# B&R Automation Studio project Panasonic_LinkaPowerCP2_A2021055 (part 35)

#### Main.st - Init, cyclic, exit code
```iecst
PROGRAM _INIT
	(* Insert code here *)

END_PROGRAM

PROGRAM _CYCLIC

	//Alarmy pracoviska č.2 (200 - 299)//
	//A200 - ST3_Zakladanie tesnenia - porucha precitania kodu paletky !!!
	//A201 - ST3_Zakladanie tesnenia - porucha precitania QR kodu !!!
	//A202 - ST3_Zakladanie tesnenia - porucha serva zdvihu !!!
	//A203 - ST3_Zakladanie tesnenia - porucha serva pojazdu !!!
	//A204 - ST3_Zakladanie tesnenia - porucha vysunutia pritlacania !!!
	//A205 - ST3_Zakladanie tesnenia - porucha zasunutia pritlacania !!!
	//A206 - ST3_Zakladanie tesnenia - narusenie optickej bariery !!!
	//A207 - ST3_Zakladanie tesnenia - bol stlaceny bumper suflika !!!
	//A208 - ST3_Zakladanie tesnenia - porucha snimaca kopita IS7 !!!
	//A209 - ST4_Maticovacka - porucha vysunutia centrovacky !!!
	//A210 - ST4_Maticovacka - porucha zasunutia centrovacky !!!
	//A211 - ST4_Maticovacka - porucha precitania kodu paletky !!!
	//A212 - ST5_Srobovanie - porucha vysunutia centrovacky !!!
	//A213 - ST5_Srobovanie - porucha zasunutia centrovacky !!!
	//A214 - ST5_Srobovanie - porucha precitania kodu paletky !!!
	//A215 - ST5_Srobovanie - porucha serva manipulatora os X !!!
	//A216 - ST5_Srobovanie - porucha serva manipulatora os Y !!!
	//A217 - ST6_Zvaranie - porucha vysunutia centrovacky !!!
	//A218 - ST6_Zvaranie - porucha zasunutia centrovacky !!!
	//A219 - ST6_Zvaranie - porucha precitania kodu paletky !!!
	//A220 - ST6_Zvaranie - porucha serva zdvihu zvarania !!!
	//A221 - ST6_Zvaranie - porucha presunu pojazdu zvarania !!!
	//A222 - ST6_Zvaranie - porucha zvaracky !!!
	//A223 - ST6_Cistenie - porucha zatvorenia dveri !!!
	//A224 - ST6_Cistenie - porucha otvorenia dveri !!!
	//A225 - ST3_Zakladanie tesnenia - CAM 1 porucha komunikacie FTP !!!
	//A226 - ST3_Zakladanie tesnenia - CAM 7 porucha komunikacie FTP !!!
	//A227 - ST3_Zakladanie tesnenia - CAM 8 porucha komunikacie FTP !!!
	//A228 - ST3_Zakladanie tesnenia - CAM 17 porucha komunikacie FTP !!!
	//A229 - ST4_Maticovacka - CAM 9 porucha komunikacie FTP !!!
	//A230 - ST3_Zakladanie tesnenia - porucha komunikacie zo serverom !!!
	//A231 - ST4_Maticovacka - porucha komunikacie zo serverom !!!
	//A232 - ST5_Srobovanie - CAM 10 porucha komunikacie FTP !!!
	//A233 - ST5_Srobovanie - porucha komunikacie zo serverom !!!
	//A234 - ST6_Zvaranie - CAM 11 porucha komunikacie FTP !!!
	//A235 - ST6_Zvaranie - CAM 12 porucha komunikacie FTP !!!
	//A236 - ST6_Zvaranie - porucha komunikacie zo serverom !!!
	//A237 - ST5_Srobovanie - skrutka M4 nieje pripravena !!!
	//A238 - ST5_Srobovanie - skrutka M5 nieje pripravena !!!
	//A239 - ST5_Srobovanie - skrutka M6 nieje pripravena !!!
	//A240 - ST4_Maticovacka - matica M4 nieje pripravena !!!
	//A241 - ST5_Srobovanie - porucha serva manipulatora os X !!!
	//A242 - ST5_Srobovanie - porucha serva manipulatora os Y !!!
	//A243 - P2_Robot - porucha napajania !!!
	//A244 - P2_Robot - nieje online !!!
	//A245 - Pracovisko 2 - Porucha tlaku vzduchu !!!
	//A246 - Pracovisko 2 - Modul DI21 nieje online !!!
	//A247 - Pracovisko 2 - Modul DI22 nieje online !!!
	//A248 - Pracovisko 2 - Modul DI23 nieje online !!!
	//A249 - Pracovisko 2 - Modul DI24 nieje online !!!
	//A250 - Pracovisko 2 - Modul DI25 nieje online !!!
	//A251 - Pracovisko 2 - Modul DM21 nieje online !!!
	//A252 - Pracovisko 2 - Modul DS21 nieje online !!!
    //A253 - Pracovisko 2 - Modul DS22 nieje online !!!
    //A254 - Pracovisko 2 - Modul DS23 nieje online !!!
	//A255 - Pracovisko 2 - Modul SI21 nieje online !!!
    //A256 - Pracovisko 2 - Modul SI22 nieje online !!!
	//A257 - Pracovisko 2 - Ventilovy termnal VT1 nieje online !!!
	//A258 - Pracovisko 2 - Ventilovy termnal VT2 nieje online !!!
    //A259 - Pracovisko 2 - Ventilovy termnal VT3 nieje online !!!
    //A260 - ST5_Srobovanie - Skrutkovacka M4 nieje online !!!
    //A261 - ST5_Srobovanie - Skrutkovacka M5 nieje online !!!
    //A262 - ST5_Srobovanie - Skrutkovacka M6 nieje online !!!
    //A263 - ST4_Maticovacka - Maticovacka M4 nieje online !!!
    //A264 - Pracovisko 2 - Kamery KAM1, KAM7, KAM10, KAM11, KAM12 a KAM17 niesu online !!!
    //A265 - Pracovisko 2 - Kamera KAM8 nieje online !!!
    //A266 - Pracovisko 2 - Kamera KAM9 nieje online !!!
    //A267 - ST4_Maticovacka - Porucha maticovacky M4 !!!
    //A268 - ST5_Srobovanie - Porucha vysunutia skrutkovacky M4 !!!
    //A269 - ST5_Srobovanie - Porucha vysunutia skrutkovacky M5 !!!
    //A270 - ST5_Srobovanie - Porucha vysunutia skrutkovacky M6 !!!
    //A271 - P2_Robot - porucha !!!
    //A272 - ST5_Srobovanie - Presiahnuty cas skrutkovania skrutky M4 !!!
    //A273 - ST5_Srobovanie - Presiahnuty cas skrutkovania skrutky M5 !!!
    //A274 - ST5_Srobovanie - Presiahnuty cas skrutkovania skrutky M6 !!!
    //A275 - ST5_Srobovanie - Skrutkovacka M4 nieje READY !!!
    //A276 - ST5_Srobovanie - Skrutkovacka M5 nieje READY !!!
    //A277 - ST5_Srobovanie - Skrutkovacka M6 nieje READY !!!
    //A278 - Pracovisko 2 - Prekrocena teplota motora vrchneho dopravnika !!!
    //A279 - Pracovisko 2 - Prekrocena teplota motora spodneho dopravnika !!!
    //A280 - Pracovisko 2 - Narusenie optickej bariery na vystupe !!!
    //A281 - Pracovisko 2 - Bolo stlacene tlacitko CS na ovladacom paneli !!!
    //A282 - Pracovisko 2 - Bolo stlacene tlacitko CS na rozvodnej skrini !!!
    //A283 - Pracovisko 2 - Bolo stlacene tlacitko CS robota !!!
    //A284 - Pracovisko 2 - Bolo stlacene tlacitko CS na dvojrucnom ovladani !!!
    //A285 - P2_Robot - Porucha odobratia Top Coveru z paletky !!!
    //A286 - ST3_Zakladanie tesnenia - Porucha vyvezenia paletky zo stopra !!!
    //A287 - ST4_Maticovacka - Porucha vyvezenia paletky zo stopra !!!
	//A288 - ST5_Srobovanie - Porucha vyvezenia paletky zo stopra !!!
    //A289 - ST6_Zvaranie - Porucha vyvezenia paletky zo stopra !!!
    //A290 - ST3_Zakladanie tesnenia - Porucha komunikacie s kamerou CAM 1 !!!
    //A291 - ST3_Zakladanie tesnenia - Porucha komunikacie s kamerou CAM 7 !!!
    //A292 - ST3_Zakladanie tesnenia - Porucha komunikacie s kamerou CAM 8 !!!
    //A293 - ST3_Zakladanie tesnenia - Porucha komunikacie s kamerou CAM 17 !!!
    //A294 - ST4_Maticovacka - Porucha komunikacie s kamerou CAM 9 !!!
    //A295 - ST5_Srobovanie - Porucha komunikacie s kamerou CAM 10 !!!
    //A296 - ST6_Zvaranie - Porucha komunikacie s kamerou CAM 11 !!!
    //A297 - ST6_Zvaranie - Porucha komunikacie s kamerou CAM 12 !!!
    //A298 - ST4_Maticovacka - Porucha pripravy matice M4 !!!
    //A299 - Akumulacny stoper - Porucha vyvezenia paletky zo stopra !!!

    //*********************Pracovisko 2 - Porucha tlaku vzduchu*********************************//
	IF CasKontroly_TlakVzduchu.Q THEN
		P2_Alarmy[245]:= TRUE;
		P2_Pracovisko.STAV.Porucha_ST1:= TRUE;
		P2_Pracovisko.STAV.Porucha_ST2:= TRUE;
		P2_Pracovisko.STAV.Porucha_ST3:= TRUE;
		P2_Pracovisko.STAV.Porucha_ST4:= TRUE;
		P2_Pracovisko.STAV.Porucha_ST5:= TRUE;
	END_IF

	IF Safety.STAV.P2_ZonaBunky_AKTIVNA AND NOT P2_Pracovisko.IN.TlakVzduchu_OK THEN
		CasKontroly_TlakVzduchu.IN:= TRUE;
	ELSE
		CasKontroly_TlakVzduchu.IN:= FALSE;
	END_IF

	CasKontroly_TlakVzduchu.PT:= T#5s;
	CasKontroly_TlakVzduchu();

	//**********************************Porucha - kamerovy systém nieje online****************************************//
	IF CasKontroly_KAMsystem.Q THEN
		P2_Alarmy[264]:= TRUE;
		P2_Pracovisko.STAV.Porucha_ST1:= TRUE;
		P2_Pracovisko.STAV.Porucha_ST2:= TRUE;
		P2_Pracovisko.STAV.Porucha_ST3:= TRUE;
		P2_Pracovisko.STAV.Porucha_ST4:= TRUE;
		P2_Pracovisko.STAV.Porucha_ST5:= TRUE;
	END_IF

	IF CasKontroly_KAM8.Q THEN
		P2_Alarmy[265]:= TRUE;
		P2_Pracovisko.STAV.Porucha_ST1:= TRUE;
	END_IF

	IF CasKontroly_KAM9.Q THEN
		P2_Alarmy[266]:= TRUE;
		P2_Pracovisko.STAV.Porucha_ST2:= TRUE;
	END_IF

	IF NOT P3_Pracovisko.IN.Kamery_ControlUnit_KomOK AND P2_Pracovisko.Automat THEN
		CasKontroly_KAMsystem.IN:= TRUE;
	ELSE
		CasKontroly_KAMsystem.IN:= FALSE;
	END_IF

	IF NOT CAM8.STAV.READY AND P2_Pracovisko.Automat THEN
		CasKontroly_KAM8.IN:= TRUE;
	ELSE
		CasKontroly_KAM8.IN:= FALSE;
	END_IF

	IF NOT CAM9.STAV.READY AND P2_Pracovisko.Automat THEN
		CasKontroly_KAM9.IN:= TRUE;
	ELSE
		CasKontroly_KAM9.IN:= FALSE;
	END_IF

	CasKontroly_KAMsystem.PT:= T#2s;
	CasKontroly_KAMsystem();
    CasKontroly_KAM8.PT:= T#2s;
	CasKontroly_KAM8();
	CasKontroly_KAM9.PT:= T#2s;
	CasKontroly_KAM9();

	//**********************************Porucha - IO moduly niesu online**************************************************//
	IF CasKontroly_Moduly.Q THEN
		P2_Alarmy[246]:= TRUE;
		P2_Pracovisko.STAV.Porucha_ST1:= TRUE;
		P2_Pracovisko.STAV.Porucha_ST2:= TRUE;
		P2_Pracovisko.STAV.Porucha_ST3:= TRUE;
		P2_Pracovisko.STAV.Porucha_ST4:= TRUE;
		P2_Pracovisko.STAV.Porucha_ST5:= TRUE;
	END_IF

	IF Safety.STAV.P2_ZonaBunky_AKTIVNA AND (NOT P2_Pracovisko.IN.ModulFesto_IO_KomOK OR NOT P2_Pracovisko.IN.ModulWeidmuller_IO_KomOK) THEN
		CasKontroly_Moduly.IN:= TRUE;
	ELSE
		CasKontroly_Moduly.IN:= FALSE;
	END_IF

	CasKontroly_Moduly.PT:= T#2s;
	CasKontroly_Moduly();

	//********************************Porucha - ventilového terminálu*********************************************//
	IF CasKontroly_VentTerminalov.Q THEN
		P2_Alarmy[257]:= TRUE;
		P2_Pracovisko.STAV.Porucha_ST1:= TRUE;
		P2_Pracovisko.STAV.Porucha_ST2:= TRUE;
		P2_Pracovisko.STAV.Porucha_ST3:= TRUE;
		P2_Pracovisko.STAV.Porucha_ST4:= TRUE;
		P2_Pracovisko.STAV.Porucha_ST5:= TRUE;
	END_IF

	IF Safety.STAV.P2_ZonaBunky_AKTIVNA AND NOT P2_Pracovisko.IN.VentilovyTerminal_KomOK THEN
		CasKontroly_VentTerminalov.IN:= TRUE;
	ELSE
		CasKontroly_VentTerminalov.IN:= FALSE;
	END_IF

	CasKontroly_VentTerminalov.PT:= T#2s;
	CasKontroly_VentTerminalov();

	//********************************Porucha - skrutkovacky niesu online**********************************************//
	IF CasKontroly_Skrutkovacky.Q THEN
		IF NOT P2_Pracovisko.IN.Skrutkovacka_M4_KomOK THEN
			P2_Alarmy[260]:= TRUE;
			P2_Pracovisko.STAV.Porucha_ST4:= TRUE;
		END_IF
		IF NOT P2_Pracovisko.IN.Skrutkovacka_M5_KomOK THEN
			P2_Alarmy[261]:= TRUE;
			P2_Pracovisko.STAV.Porucha_ST4:= TRUE;
		END_IF
		IF NOT P2_Pracovisko.IN.Skrutkovacka_M6_KomOK THEN
			P2_Alarmy[262]:= TRUE;
			P2_Pracovisko.STAV.Porucha_ST4:= TRUE;
		END_IF
		IF NOT P2_Pracovisko.IN.Maticovacka_M4_KomOK THEN
			P2_Alarmy[263]:= TRUE;
			P2_Pracovisko.STAV.Porucha_ST2:= TRUE;
		END_IF
	END_IF

	IF Safety.STAV.P2_ZonaBunky_AKTIVNA AND
		(NOT P2_Pracovisko.IN.Skrutkovacka_M4_KomOK OR
		NOT P2_Pracovisko.IN.Skrutkovacka_M5_KomOK OR
		NOT P2_Pracovisko.IN.Skrutkovacka_M6_KomOK OR
		NOT P2_Pracovisko.IN.Maticovacka_M4_KomOK) THEN
		CasKontroly_Skrutkovacky.IN:= TRUE;
	ELSE
		CasKontroly_Skrutkovacky.IN:= FALSE;
	END_IF

	CasKontroly_Skrutkovacky.PT:= T#2s;
	CasKontroly_Skrutkovacky();

	//*********************************Porucha - robot nieje online************************************************//
	IF CasKontroly_Robota.Q THEN
		P2_Alarmy[244]:= TRUE;
		P2_Pracovisko.STAV.Porucha_ST4:= TRUE;
		P2_Pracovisko.STAV.Porucha_ST5:= TRUE;
	END_IF

	IF Safety.STAV.P2_ZonaBunky_AKTIVNA AND NOT P2_Pracovisko.IN.Robot_KomOK THEN
		CasKontroly_Robota.IN:= TRUE;
	ELSE
		CasKontroly_Robota.IN:= FALSE;
	END_IF

	CasKontroly_Robota.PT:= T#2s;
	CasKontroly_Robota();

	//********************Pracovisko 2 - Porucha ochrannej bariéry zdvihu zakladača tesnenia****************************************//
	IF CasKontroly_BarieryZakladaca.Q THEN
		P2_Alarmy[206]:= TRUE;
		P2_Pracovisko.STAV.Porucha_ST1:= TRUE;
	END_IF

    CasKontroly_BarieryZakladaca.IN:= P2_ZakladacTesnenia.Automat AND NOT Safety.STAV.P2_ZaklTesn_Bariera_AKTIVNA AND Safety.STAV.P2_ZaklTesn_PojazdMuting_AKTIVNY;
	CasKontroly_BarieryZakladaca.PT:= T#2s;
	CasKontroly_BarieryZakladaca();

	//*********************Pracovisko 2 - Porucha serva zdvihu zakladača tesnenia***************//
	IF CasPoruchyServaZdvihuZakladaca.Q THEN
		P2_Alarmy[202]:= TRUE;
		P2_Pracovisko.STAV.Porucha_ST1:= TRUE;
	END_IF

	IF Safety.STAV.P2_ZonaZakladacaZdvih_AKTIVNA AND P2_ZakladacTesnenia.ServoZdvihuZakladaca.Status.Error THEN
		CasPoruchyServaZdvihuZakladaca.IN:= TRUE;
	ELSE
		CasPoruchyServaZdvihuZakladaca.IN:= FALSE;
	END_IF

	CasPoruchyServaZdvihuZakladaca.PT:= T#2s;
	CasPoruchyServaZdvihuZakladaca();

	//********************Pracovisko 2 - Porucha bumpera suflíka zakladača tesnenia****************************************//
	IF P2_ZakladacTesnenia.Automat AND NOT Safety.STAV.P2_ZaklTesn_Bumper_AKTIVNY THEN
		P2_Alarmy[207]:= TRUE;
		P2_Pracovisko.STAV.Porucha_ST1:= TRUE;
	END_IF

	//*********************Pracovisko 2 - Porucha serva pojazdu zakladača tesnenia***************//
	IF CasPoruchyServaPojazduZakladaca.Q THEN
		P2_Alarmy[203]:= TRUE;
		P2_Pracovisko.STAV.Porucha_ST1:= TRUE;
	END_IF

	IF Safety.STAV.P2_ZonaZakladacaPojazd_AKTIVNA AND P2_ZakladacTesnenia.ServoPojazduZakladaca.Status.Error THEN
		CasPoruchyServaPojazduZakladaca.IN:= TRUE;
	ELSE
		CasPoruchyServaPojazduZakladaca.IN:= FALSE;
	END_IF

	CasPoruchyServaPojazduZakladaca.PT:= T#2s;
	CasPoruchyServaPojazduZakladaca();

	//*********************Pracovisko 2 - Porucha serva manipulatora šrobovania os X***************//
	IF CasPoruchyServaSrobovaniaOsX.Q THEN
		P2_Alarmy[215]:= TRUE;
		P2_Pracovisko.STAV.Porucha_ST4:= TRUE;
	END_IF

	IF Safety.STAV.P2_ZonaBunky_AKTIVNA AND P2_Srobovanie.ServoManipulOsX.Status.Error THEN
		CasPoruchyServaSrobovaniaOsX.IN:= TRUE;
	ELSE
		CasPoruchyServaSrobovaniaOsX.IN:= FALSE;
	END_IF

	CasPoruchyServaSrobovaniaOsX.PT:= T#2s;
	CasPoruchyServaSrobovaniaOsX();

	//*********************Pracovisko 2 - Porucha serva manipulatora šrobovania os Y***************//
	IF CasPoruchyServaSrobovaniaOsY.Q THEN
		P2_Alarmy[216]:= TRUE;
		P2_Pracovisko.STAV.Porucha_ST4:= TRUE;
	END_IF

	IF Safety.STAV.P2_ZonaBunky_AKTIVNA AND P2_Srobovanie.ServoManipulOsY.Status.Error THEN
		CasPoruchyServaSrobovaniaOsY.IN:= TRUE;
	ELSE
		CasPoruchyServaSrobovaniaOsY.IN:= FALSE;
	END_IF

	CasPoruchyServaSrobovaniaOsY.PT:= T#2s;
	CasPoruchyServaSrobovaniaOsY();

	//*********************Pracovisko 2 - Porucha serva manipulatora šrobovania os Z M4***************//
	IF CasPoruchyServaSrobovaniaOsZ_M4.Q THEN
		P2_Alarmy[247]:= TRUE;
		P2_Pracovisko.STAV.Porucha_ST4:= TRUE;
	END_IF

	IF Safety.STAV.P1_ZonaBunky_AKTIVNA AND P1_Srobovanie.ServoManipulOsZ_M4.Status.Error THEN
		CasPoruchyServaSrobovaniaOsZ_M4.IN:= TRUE;
	ELSE
		CasPoruchyServaSrobovaniaOsZ_M4.IN:= FALSE;
	END_IF

	CasPoruchyServaSrobovaniaOsZ_M4.PT:= T#2s;
	CasPoruchyServaSrobovaniaOsZ_M4();

	//**********************Pracovisko 2 - Porucha serva zdvihu zvarania****************************//
	IF CasPoruchyServaZdvihuZvarania.Q THEN
		P2_Alarmy[220]:= TRUE;
		P2_Pracovisko.STAV.Porucha_ST5:= TRUE;
	END_IF

	IF Safety.STAV.P2_ZonaBunky_AKTIVNA AND P2_Zvaranie.ServoZdvihuZvarania.Status.Error THEN
		CasPoruchyServaZdvihuZvarania.IN:= TRUE;
	ELSE
		CasPoruchyServaZdvihuZvarania.IN:= FALSE;
	END_IF

	CasPoruchyServaZdvihuZvarania.PT:= T#2s;
	CasPoruchyServaZdvihuZvarania();

	//********************Pracovisko 2 - Porucha skrutkovacieho setu M4******************************//
	IF P2_Srobovanie.Automat AND P2_Srobovanie.SkrutSet_M4.STAV.ERROR THEN
		P2_Alarmy[248]:= TRUE;
		P2_Pracovisko.STAV.Porucha_ST4:= TRUE;
	END_IF

	//********************Pracovisko 2 - Porucha skrutkovacieho setu matice M4******************************//
	IF P2_StoperMaticovacky.Automat AND P2_StoperMaticovacky.SkrutSet_MaticaM4.STAV.ERROR THEN
		P2_Alarmy[249]:= TRUE;
		P2_Pracovisko.STAV.Porucha_ST2:= TRUE;
	END_IF

	//****************************Pracovisko 2 - porucha vrchného dopravníka**********************************//
	IF NOT P2_Dopravniky.IN.TeplotaMotoraDopravBunky_OK AND P2_Pracovisko.STAV.Automat THEN
		P2_Alarmy[278]:= TRUE;
		P2_Pracovisko.STAV.Porucha_ST1:= TRUE;
		P2_Pracovisko.STAV.Porucha_ST2:= TRUE;
		P2_Pracovisko.STAV.Porucha_ST3:= TRUE;
		P2_Pracovisko.STAV.Porucha_ST4:= TRUE;
		P2_Pracovisko.STAV.Porucha_ST5:= TRUE;
	END_IF

	//*****************************Pracovisko 2 - porucha spodného dopravníka************************************//
	IF NOT P2_Dopravniky.IN.TeplotaMotoraVratnehoDoprav_OK AND P2_Pracovisko.STAV.Automat THEN
		P2_Alarmy[279]:= TRUE;
	END_IF

	//******************************Pracovisko 2 - narušenie výstupnej bariery***********************************//
	IF NOT Safety.STAV.P3_Bunka_VstupBariera_AKTIVNA AND NOT Safety.STAV.P3_Bunka_Zamky_AKTIVNE AND NOT Safety.STAV.P3_VyblokovanieZamkov_AKTIVNE AND P2_Pracovisko.STAV.Automat THEN
		P2_Alarmy[280]:= TRUE;
		P2_Pracovisko.STAV.Porucha_ST2:= TRUE;
		P2_Pracovisko.STAV.Porucha_ST3:= TRUE;
		P2_Pracovisko.STAV.Porucha_ST4:= TRUE;
		P2_Pracovisko.STAV.Porucha_ST5:= TRUE;
	END_IF

	//******************************Stlačenie tlačítok CS*******************************************************//
	IF EDGENEG(Safety.STAV.P2_Panel_TlacitkoCS_ODBLOK) THEN
		P2_Alarmy[281]:= TRUE;
	END_IF

	IF EDGENEG(Safety.STAV.P2_Rozvadzac_TlacitkoCS_ODBLOK) THEN
		P2_Alarmy[282]:= TRUE;
	END_IF

	IF EDGENEG(Safety.STAV.P2_Robot_TlacitkoCS_ODBLOK) THEN
		P2_Alarmy[283]:= TRUE;
	END_IF

	IF EDGENEG(Safety.STAV.P2_DvojrucOvl_TlacitkoCS_ODBLOK) THEN
		P2_Alarmy[284]:= TRUE;
	END_IF

	//***************************************************Nasetovanie alarmov****************************************************//

	IF P2_Alarmy[200] THEN
		MpAlarmXSet(gAlarmXCore, 'A200');
	ELSE
		MpAlarmXReset(gAlarmXCore, 'A200');
	END_IF

	IF P2_Alarmy[201] THEN
		MpAlarmXSet(gAlarmXCore, 'A201');
	ELSE
		MpAlarmXReset(gAlarmXCore, 'A201');
	END_IF

	IF P2_Alarmy[202] THEN
		MpAlarmXSet(gAlarmXCore, 'A202');
	ELSE
		MpAlarmXReset(gAlarmXCore, 'A202');
	END_IF

	IF P2_Alarmy[203] THEN
		MpAlarmXSet(gAlarmXCore, 'A203');
	ELSE
		MpAlarmXReset(gAlarmXCore, 'A203');
	END_IF

	IF P2_Alarmy[204] THEN
		MpAlarmXSet(gAlarmXCore, 'A204');
	ELSE
		MpAlarmXReset(gAlarmXCore, 'A204');
	END_IF

	IF P2_Alarmy[205] THEN
		MpAlarmXSet(gAlarmXCore, 'A205');
	ELSE
		MpAlarmXReset(gAlarmXCore, 'A205');
	END_IF

	IF P2_Alarmy[206] THEN
		MpAlarmXSet(gAlarmXCore, 'A206');
	ELSE
		MpAlarmXReset(gAlarmXCore, 'A206');
	END_IF

	IF P2_Alarmy[207] THEN
		MpAlarmXSet(gAlarmXCore, 'A207');
	ELSE
		MpAlarmXReset(gAlarmXCore, 'A207');
	END_IF

	IF P2_Alarmy[208] THEN
		MpAlarmXSet(gAlarmXCore, 'A208');
	ELSE
		MpAlarmXReset(gAlarmXCore, 'A208');
	END_IF

	IF P2_Alarmy[209] THEN
		MpAlarmXSet(gAlarmXCore, 'A209');
	ELSE
		MpAlarmXReset(gAlarmXCore, 'A209');
	END_IF

	IF P2_Alarmy[210] THEN
		MpAlarmXSet(gAlarmXCore, 'A210');
	ELSE
		MpAlarmXReset(gAlarmXCore, 'A210');
	END_IF

	IF P2_Alarmy[211] THEN
		MpAlarmXSet(gAlarmXCore, 'A211');
	ELSE
		MpAlarmXReset(gAlarmXCore, 'A211');
	END_IF

	IF P2_Alarmy[212] THEN
		MpAlarmXSet(gAlarmXCore, 'A212');
	ELSE
		MpAlarmXReset(gAlarmXCore, 'A212');
	END_IF

	IF P2_Alarmy[213] THEN
		MpAlarmXSet(gAlarmXCore, 'A213');
	ELSE
		MpAlarmXReset(gAlarmXCore, 'A213');
	END_IF

	IF P2_Alarmy[214] THEN
		MpAlarmXSet(gAlarmXCore, 'A214');
	ELSE
		MpAlarmXReset(gAlarmXCore, 'A214');
	END_IF

	IF P2_Alarmy[215] THEN
		MpAlarmXSet(gAlarmXCore, 'A215');
	ELSE
		MpAlarmXReset(gAlarmXCore, 'A215');
	END_IF

	IF P2_Alarmy[216] THEN
		MpAlarmXSet(gAlarmXCore, 'A216');
	ELSE
		MpAlarmXReset(gAlarmXCore, 'A216');
	END_IF

	IF P2_Alarmy[217] THEN
		MpAlarmXSet(gAlarmXCore, 'A217');
	ELSE
		MpAlarmXReset(gAlarmXCore, 'A217');
	END_IF

	IF P2_Alarmy[218] THEN
		MpAlarmXSet(gAlarmXCore, 'A218');
	ELSE
		MpAlarmXReset(gAlarmXCore, 'A218');
	END_IF

	IF P2_Alarmy[219] THEN
		MpAlarmXSet(gAlarmXCore, 'A219');
	ELSE
		MpAlarmXReset(gAlarmXCore, 'A219');
	END_IF

	IF P2_Alarmy[220] THEN
		MpAlarmXSet(gAlarmXCore, 'A220');
	ELSE
		MpAlarmXReset(gAlarmXCore, 'A220');
	END_IF

	IF P2_Alarmy[221] THEN
		MpAlarmXSet(gAlarmXCore, 'A221');
	ELSE
		MpAlarmXReset(gAlarmXCore, 'A221');
	END_IF

	IF P2_Alarmy[222] THEN
		MpAlarmXSet(gAlarmXCore, 'A222');
	ELSE
		MpAlarmXReset(gAlarmXCore, 'A222');
	END_IF

	IF P2_Alarmy[223] THEN
		MpAlarmXSet(gAlarmXCore, 'A223');
	ELSE
		MpAlarmXReset(gAlarmXCore, 'A223');
	END_IF

	IF P2_Alarmy[224] THEN
		MpAlarmXSet(gAlarmXCore, 'A224');
	ELSE
		MpAlarmXReset(gAlarmXCore, 'A224');
	END_IF

	IF P2_Alarmy[225] THEN
		MpAlarmXSet(gAlarmXCore, 'A225');
	ELSE
		MpAlarmXReset(gAlarmXCore, 'A225');
	END_IF

	IF P2_Alarmy[226] THEN
		MpAlarmXSet(gAlarmXCore, 'A226');
	ELSE
		MpAlarmXReset(gAlarmXCore, 'A226');
	END_IF

	IF P2_Alarmy[227] THEN
		MpAlarmXSet(gAlarmXCore, 'A227');
	ELSE
		MpAlarmXReset(gAlarmXCore, 'A227');
	END_IF

	IF P2_Alarmy[228] THEN
		MpAlarmXSet(gAlarmXCore, 'A228');
	ELSE
		MpAlarmXReset(gAlarmXCore, 'A228');
	END_IF

	IF P2_Alarmy[229] THEN
		MpAlarmXSet(gAlarmXCore, 'A229');
	ELSE
		MpAlarmXReset(gAlarmXCore, 'A229');
	END_IF

	IF P2_Alarmy[230] THEN
		MpAlarmXSet(gAlarmXCore, 'A230');
	ELSE
		MpAlarmXReset(gAlarmXCore, 'A230');
	END_IF

	IF P2_Alarmy[231] THEN
		MpAlarmXSet(gAlarmXCore, 'A231');
	ELSE
		MpAlarmXReset(gAlarmXCore, 'A231');
	END_IF

	IF P2_Alarmy[232] THEN
		MpAlarmXSet(gAlarmXCore, 'A232');
	ELSE
		MpAlarmXReset(gAlarmXCore, 'A232');
	END_IF

	IF P2_Alarmy[233] THEN
		MpAlarmXSet(gAlarmXCore, 'A233');
	ELSE
		MpAlarmXReset(gAlarmXCore, 'A233');
	END_IF

	IF P2_Alarmy[234] THEN
		MpAlarmXSet(gAlarmXCore, 'A234');
	ELSE
		MpAlarmXReset(gAlarmXCore, 'A234');
	END_IF

	IF P2_Alarmy[235] THEN
		MpAlarmXSet(gAlarmXCore, 'A235');
	ELSE
		MpAlarmXReset(gAlarmXCore, 'A235');
	END_IF

	IF P2_Alarmy[236] THEN
		MpAlarmXSet(gAlarmXCore, 'A236');
	ELSE
		MpAlarmXReset(gAlarmXCore, 'A236');
	END_IF

	IF P2_Alarmy[237] THEN
		MpAlarmXSet(gAlarmXCore, 'A237');
	ELSE
		MpAlarmXReset(gAlarmXCore, 'A237');
	END_IF

	IF P2_Alarmy[238] THEN
		MpAlarmXSet(gAlarmXCore, 'A238');
	ELSE
		MpAlarmXReset(gAlarmXCore, 'A238');
	END_IF

	IF P2_Alarmy[239] THEN
		MpAlarmXSet(gAlarmXCore, 'A239');
	ELSE
		MpAlarmXReset(gAlarmXCore, 'A239');
	END_IF

	IF P2_Alarmy[240] THEN
		MpAlarmXSet(gAlarmXCore, 'A240');
	ELSE
		MpAlarmXReset(gAlarmXCore, 'A240');
	END_IF

	IF P2_Alarmy[241] THEN
		MpAlarmXSet(gAlarmXCore, 'A241');
	ELSE
		MpAlarmXReset(gAlarmXCore, 'A241');
	END_IF

	IF P2_Alarmy[242] THEN
		MpAlarmXSet(gAlarmXCore, 'A242');
	ELSE
		MpAlarmXReset(gAlarmXCore, 'A242');
	END_IF

	IF P2_Alarmy[243] THEN
		MpAlarmXSet(gAlarmXCore, 'A243');
	ELSE
		MpAlarmXReset(gAlarmXCore, 'A243');
	END_IF

	IF P2_Alarmy[244] THEN
		MpAlarmXSet(gAlarmXCore, 'A244');
	ELSE
		MpAlarmXReset(gAlarmXCore, 'A244');
	END_IF

	IF P2_Alarmy[245] THEN
		MpAlarmXSet(gAlarmXCore, 'A245');
	ELSE
		MpAlarmXReset(gAlarmXCore, 'A245');
	END_IF

	IF P2_Alarmy[246] THEN
		MpAlarmXSet(gAlarmXCore, 'A246');
	ELSE
		MpAlarmXReset(gAlarmXCore, 'A246');
	END_IF

	IF P2_Alarmy[247] THEN
		MpAlarmXSet(gAlarmXCore, 'A247');
	ELSE
		MpAlarmXReset(gAlarmXCore, 'A247');
	END_IF

	IF P2_Alarmy[248] THEN
		MpAlarmXSet(gAlarmXCore, 'A248');
	ELSE
		MpAlarmXReset(gAlarmXCore, 'A248');
	END_IF

	IF P2_Alarmy[249] THEN
		MpAlarmXSet(gAlarmXCore, 'A249');
	ELSE
		MpAlarmXReset(gAlarmXCore, 'A249');
	END_IF

	IF P2_Alarmy[250] THEN
		MpAlarmXSet(gAlarmXCore, 'A250');
	ELSE
		MpAlarmXReset(gAlarmXCore, 'A250');
	END_IF

	IF P2_Alarmy[251] THEN
		MpAlarmXSet(gAlarmXCore, 'A251');
	ELSE
		MpAlarmXReset(gAlarmXCore, 'A251');
	END_IF

	IF P2_Alarmy[252] THEN
		MpAlarmXSet(gAlarmXCore, 'A252');
	ELSE
		MpAlarmXReset(gAlarmXCore, 'A252');
	END_IF

	IF P2_Alarmy[253] THEN
		MpAlarmXSet(gAlarmXCore, 'A253');
	ELSE
		MpAlarmXReset(gAlarmXCore, 'A253');
	END_IF

	IF P2_Alarmy[254] THEN
		MpAlarmXSet(gAlarmXCore, 'A254');
	ELSE
		MpAlarmXReset(gAlarmXCore, 'A254');
	END_IF

	IF P2_Alarmy[255] THEN
		MpAlarmXSet(gAlarmXCore, 'A255');
	ELSE
		MpAlarmXReset(gAlarmXCore, 'A255');
	END_IF

	IF P2_Alarmy[256] THEN
		MpAlarmXSet(gAlarmXCore, 'A256');
	ELSE
		MpAlarmXReset(gAlarmXCore, 'A256');
	END_IF

	IF P2_Alarmy[257] THEN
		MpAlarmXSet(gAlarmXCore, 'A257');
	ELSE
		MpAlarmXReset(gAlarmXCore, 'A257');
	END_IF

	IF P2_Alarmy[258] THEN
		MpAlarmXSet(gAlarmXCore, 'A258');
	ELSE
		MpAlarmXReset(gAlarmXCore, 'A258');
	END_IF

	IF P2_Alarmy[259] THEN
		MpAlarmXSet(gAlarmXCore, 'A259');
	ELSE
		MpAlarmXReset(gAlarmXCore, 'A259');
	END_IF

	IF P2_Alarmy[260] THEN
		MpAlarmXSet(gAlarmXCore, 'A260');
	ELSE
		MpAlarmXReset(gAlarmXCore, 'A260');
	END_IF

	IF P2_Alarmy[261] THEN
		MpAlarmXSet(gAlarmXCore, 'A261');
	ELSE
		MpAlarmXReset(gAlarmXCore, 'A261');
	END_IF

	IF P2_Alarmy[262] THEN
		MpAlarmXSet(gAlarmXCore, 'A262');
	ELSE
		MpAlarmXReset(gAlarmXCore, 'A262');
	END_IF

	IF P2_Alarmy[263] THEN
		MpAlarmXSet(gAlarmXCore, 'A263');
	ELSE
		MpAlarmXReset(gAlarmXCore, 'A263');
	END_IF

	IF P2_Alarmy[264] THEN
		MpAlarmXSet(gAlarmXCore, 'A264');
	ELSE
		MpAlarmXReset(gAlarmXCore, 'A264');
	END_IF

	IF P2_Alarmy[265] THEN
		MpAlarmXSet(gAlarmXCore, 'A265');
	ELSE
		MpAlarmXReset(gAlarmXCore, 'A265');
	END_IF

	IF P2_Alarmy[266] THEN
		MpAlarmXSet(gAlarmXCore, 'A266');
	ELSE
		MpAlarmXReset(gAlarmXCore, 'A266');
	END_IF

	IF P2_Alarmy[267] THEN
		MpAlarmXSet(gAlarmXCore, 'A267');
	ELSE
		MpAlarmXReset(gAlarmXCore, 'A267');
	END_IF

	IF P2_Alarmy[268] THEN
		MpAlarmXSet(gAlarmXCore, 'A268');
	ELSE
		MpAlarmXReset(gAlarmXCore, 'A268');
	END_IF

	IF P2_Alarmy[269] THEN
		MpAlarmXSet(gAlarmXCore, 'A269');
	ELSE
		MpAlarmXReset(gAlarmXCore, 'A269');
	END_IF

	IF P2_Alarmy[270] THEN
		MpAlarmXSet(gAlarmXCore, 'A270');
	ELSE
		MpAlarmXReset(gAlarmXCore, 'A270');
	END_IF

	IF P2_Alarmy[271] THEN
		MpAlarmXSet(gAlarmXCore, 'A271');
	ELSE
		MpAlarmXReset(gAlarmXCore, 'A271');
	END_IF

	IF P2_Alarmy[272] THEN
		MpAlarmXSet(gAlarmXCore, 'A272');
	ELSE
		MpAlarmXReset(gAlarmXCore, 'A272');
	END_IF

	IF P2_Alarmy[273] THEN
		MpAlarmXSet(gAlarmXCore, 'A273');
	ELSE
		MpAlarmXReset(gAlarmXCore, 'A273');
	END_IF

	IF P2_Alarmy[274] THEN
		MpAlarmXSet(gAlarmXCore, 'A274');
	ELSE
		MpAlarmXReset(gAlarmXCore, 'A274');
	END_IF

	IF P2_Alarmy[275] THEN
		MpAlarmXSet(gAlarmXCore, 'A275');
	ELSE
		MpAlarmXReset(gAlarmXCore, 'A275');
	END_IF

	IF P2_Alarmy[276] THEN
		MpAlarmXSet(gAlarmXCore, 'A276');
	ELSE
		MpAlarmXReset(gAlarmXCore, 'A276');
	END_IF

	IF P2_Alarmy[277] THEN
		MpAlarmXSet(gAlarmXCore, 'A277');
	ELSE
		MpAlarmXReset(gAlarmXCore, 'A277');
	END_IF

	IF P2_Alarmy[278] THEN
		MpAlarmXSet(gAlarmXCore, 'A278');
	ELSE
		MpAlarmXReset(gAlarmXCore, 'A278');
	END_IF

	IF P2_Alarmy[279] THEN
		MpAlarmXSet(gAlarmXCore, 'A279');
	ELSE
		MpAlarmXReset(gAlarmXCore, 'A279');
	END_IF

	IF P2_Alarmy[280] THEN
		MpAlarmXSet(gAlarmXCore, 'A280');
	ELSE
		MpAlarmXReset(gAlarmXCore, 'A280');
	END_IF

	IF P2_Alarmy[281] THEN
		MpAlarmXSet(gAlarmXCore, 'A281');
	ELSE
		MpAlarmXReset(gAlarmXCore, 'A281');
	END_IF

	IF P2_Alarmy[282] THEN
		MpAlarmXSet(gAlarmXCore, 'A282');
	ELSE
		MpAlarmXReset(gAlarmXCore, 'A282');
	END_IF

	IF P2_Alarmy[283] THEN
		MpAlarmXSet(gAlarmXCore, 'A283');
	ELSE
		MpAlarmXReset(gAlarmXCore, 'A283');
	END_IF

	IF P2_Alarmy[284] THEN
		MpAlarmXSet(gAlarmXCore, 'A284');
	ELSE
		MpAlarmXReset(gAlarmXCore, 'A284');
	END_IF

	IF P2_Alarmy[285] THEN
		MpAlarmXSet(gAlarmXCore, 'A285');
	ELSE
		MpAlarmXReset(gAlarmXCore, 'A285');
	END_IF

	IF P2_Alarmy[286] THEN
		MpAlarmXSet(gAlarmXCore, 'A286');
	ELSE
		MpAlarmXReset(gAlarmXCore, 'A286');
	END_IF

	IF P2_Alarmy[287] THEN
		MpAlarmXSet(gAlarmXCore, 'A287');
	ELSE
		MpAlarmXReset(gAlarmXCore, 'A287');
	END_IF

	IF P2_Alarmy[288] THEN
		MpAlarmXSet(gAlarmXCore, 'A288');
	ELSE
		MpAlarmXReset(gAlarmXCore, 'A288');
	END_IF

	IF P2_Alarmy[289] THEN
		MpAlarmXSet(gAlarmXCore, 'A289');
	ELSE
		MpAlarmXReset(gAlarmXCore, 'A289');
	END_IF

	IF P2_Alarmy[290] THEN
		MpAlarmXSet(gAlarmXCore, 'A290');
	ELSE
		MpAlarmXReset(gAlarmXCore, 'A290');
	END_IF

	IF P2_Alarmy[291] THEN
		MpAlarmXSet(gAlarmXCore, 'A291');
	ELSE
		MpAlarmXReset(gAlarmXCore, 'A291');
	END_IF

	IF P2_Alarmy[292] THEN
		MpAlarmXSet(gAlarmXCore, 'A292');
	ELSE
		MpAlarmXReset(gAlarmXCore, 'A292');
	END_IF

	IF P2_Alarmy[293] THEN
		MpAlarmXSet(gAlarmXCore, 'A293');
	ELSE
		MpAlarmXReset(gAlarmXCore, 'A293');
	END_IF

	IF P2_Alarmy[294] THEN
		MpAlarmXSet(gAlarmXCore, 'A294');
	ELSE
		MpAlarmXReset(gAlarmXCore, 'A294');
	END_IF

	IF P2_Alarmy[295] THEN
		MpAlarmXSet(gAlarmXCore, 'A295');
	ELSE
		MpAlarmXReset(gAlarmXCore, 'A295');
	END_IF

	IF P2_Alarmy[296] THEN
		MpAlarmXSet(gAlarmXCore, 'A296');
	ELSE
		MpAlarmXReset(gAlarmXCore, 'A296');
	END_IF

	IF P2_Alarmy[297] THEN
		MpAlarmXSet(gAlarmXCore, 'A297');
	ELSE
		MpAlarmXReset(gAlarmXCore, 'A297');
	END_IF

	IF P2_Alarmy[298] THEN
		MpAlarmXSet(gAlarmXCore, 'A298');
	ELSE
		MpAlarmXReset(gAlarmXCore, 'A298');
	END_IF

	IF P2_Alarmy[299] THEN
		MpAlarmXSet(gAlarmXCore, 'A299');
	ELSE
		MpAlarmXReset(gAlarmXCore, 'A299');
	END_IF

	//*************************************Potvrdenie alarmov*********************************************************//
	IF P2_AlarmyVizu.PotvrdAlarmy THEN
		brsmemset(ADR(P2_Alarmy),0,SIZEOF(P2_Alarmy));
		P2_Pracovisko.STAV.Porucha_ST1:= FALSE;
		P2_Pracovisko.STAV.Porucha_ST2:= FALSE;
		P2_Pracovisko.STAV.Porucha_ST3:= FALSE;
		P2_Pracovisko.STAV.Porucha_ST4:= FALSE;
		P2_Pracovisko.STAV.Porucha_ST5:= FALSE;
		IF NOT P2_Srobovanie.Automat THEN
			P2_Srobovanie.ServoManipulOsX.Command.ErrReset:= TRUE;
			P2_Srobovanie.ServoManipulOsY.Command.ErrReset:= TRUE;
			P2_Srobovanie.ServoManipulOsZ_M4.Command.ErrReset:= TRUE;
			P2_Srobovanie.SkrutSet_M4.CMD.ResetPoruchy:= TRUE;
		END_IF
		IF NOT P2_StoperMaticovacky.Automat THEN
			P2_StoperMaticovacky.SkrutSet_MaticaM4.CMD.ResetPoruchy:= TRUE;
		END_IF
		P2_AlarmyVizu.PotvrdAlarmy:= FALSE;
	END_IF

END_PROGRAM

PROGRAM _EXIT
	(* Insert code here *)

END_PROGRAM
```

#### Variables.var - Local variables
```iecst
VAR
	i : UINT;
	CasKontroly_TlakVzduchu : TON;
	CasKontroly_KAMsystem : TON;
	CasKontroly_Moduly : TON;
	CasKontroly_VentTerminalov : TON;
	CasKontroly_Skrutkovacky : TON;
	CasKontroly_Robota : TON;
	CasPoruchyServaZdvihuZakladaca : TON;
	CasPoruchyServaPojazduZakladaca : TON;
	CasPoruchyServaSrobovaniaOsX : TON;
	CasPoruchyServaSrobovaniaOsY : TON;
	CasPoruchyServaZdvihuZvarania : TON;
	CasResetServaZdvihuZakladaca : TON;
	CasResetServaPojazduZakladaca : TON;
	CasResetovaniaServaSrobovaniaOsX : TON;
	CasResetovaniaServaSrobovaniaOsY : TON;
	CasResetServaZdvihuZvarania : TON;
	a : INT;
	CasKontroly_KAM8 : TON;
	CasKontroly_KAM9 : TON;
	CasPoruchyServaSrobovaniaOsZ_M4 : TON;
	CasKontroly_BarieryZakladaca : TON;
END_VAR
```

### Program Logical/Alarmy/P34_Alarmy (IEC)

#### Main.st - Init, cyclic, exit code
```iecst
PROGRAM _INIT
	(* Insert code here *)

END_PROGRAM

PROGRAM _CYCLIC

	//Alarmy pracoviska č.3 (300 - 399)//
	//A300 - ST7_Srobovanie - porucha vysunutia centrovacky !!!
	//A301 - ST7_Srobovanie - porucha zasunutia centrovacky !!!
	//A302 - ST8A_Leakage test A - porucha vysunutia centrovacky !!!
	//A303 - ST8A_Leakage test A - porucha zasunutia centrovacky !!!
	//A304 - ST8B_Leakage test B - porucha vysunutia centrovacky !!!
	//A305 - ST8B_Leakage test B - porucha zasunutia centrovacky !!!
	//A306 - ST8A_Leakage test A - porucha vysunutia pritlaku !!!
	//A307 - ST8A_Leakage test A - porucha zasunutia pritlaku !!!
	//A308 - ST8B_Leakage test B - porucha vysunutia pritlaku !!!
	//A309 - ST8B_Leakage test B - porucha zasunutia pritlaku !!!
	//A310 - ST8A_Leakage test A - porucha precitania kodu paletky !!!
	//A311 - ST8A_Leakage test A - porucha komunikacie zo serverom !!!
	//A312 - ST8B_Leakage test B - porucha precitania kodu paletky !!!
	//A313 - ST8B_Leakage test B - porucha komunikacie zo serverom !!!
	//A314 - ST8A_Leakage test A - je zalozeny nespravny typ spodneho kopita !!!
	//A315 - ST8B_Leakage test B - je zalozeny nespravny typ spodneho kopita !!!
	//A316 - ST7_Srobovanie - porucha vysunutia kontaktov HV testu !!!
	//A317 - ST7_Srobovanie - porucha zasunutia kontaktov HV testu !!!
	//A318 - ST7_Srobovanie - porucha vysunutia HV testu !!!
	//A319 - ST7_Srobovanie - porucha zasunutia HV testu !!!
	//A320 - ST7_Srobovanie - CAM 13 porucha komunikacie FTP !!!
	//A321 - ST7_Srobovanie - porucha precitania kodu paletky !!!
	//A322 - ST7_Srobovanie - porucha serva manipulatora os Y !!!
	//A323 - Pracovisko 3 - Porucha tlaku vzduchu !!!
	//A324 - ST7_Srobovanie - Skrutkovacka M5 nieje online !!!
	//A325 - ST7_Srobovanie - porucha komunikacie zo serverom !!!
	//A326 - ST7_HV Test - je zalozeny nespravny typ spodneho kopita !!!
    //A327 - ST7_Srobovanie - skrutka M5 nieje pripravena !!!
    //A328 - ST7_Srobovanie - skrutka K40 nieje pripravena !!!
	//A329 - ST7_Srobovanie - Skrutkovacka K40 nieje online !!!
    //A330 - ST7_Srobovanie - Kamera KAM13 nieje online !!!
    //A331 - Pracovisko 3 - Modul DI31 nieje online !!!
    //A332 - Pracovisko 3 - Modul DI32 nieje online !!!
    //A333 - Pracovisko 3 - Modul DI33 nieje online !!!
    //A334 - Pracovisko 3 - Modul DI34 nieje online !!!
    //A335 - Pracovisko 3 - Modul DM31 nieje online !!!
    //A336 - Pracovisko 3 - Modul DS31 nieje online !!!
    //A337 - Pracovisko 3 - Modul DS32 nieje online !!!
    //A338 - Pracovisko 3 - Modul DS33 nieje online !!!
    //A339 - Pracovisko 3 - Modul SI31 nieje online !!!
    //A340 - Pracovisko 3 - Ventilovy termnal VT6 nieje online !!!
	//A341 - Pracovisko 3 - Ventilovy termnal VT7 nieje online !!!
    //A342 - ST7_Srobovanie - Porucha vysunutia skrutkovacky K40 !!!
    //A343 - ST7_Srobovanie - Porucha vysunutia skrutkovacky M5 !!!
    //A344 - ST7_Srobovanie - Skrutkovacka K40 nieje READY !!!
    //A345 - ST7_Srobovanie - Skrutkovacka M5 nieje READY !!!
    //A346 - ST7_Srobovanie - Presiahnuty cas skrutkovania skrutky K40 !!!
    //A347 - ST7_Srobovanie - Presiahnuty cas skrutkovania skrutky M5 !!!
    //A348 - Pracovisko 3 - Prekrocena teplota motora vrchneho dopravnika !!!
    //A349 - Pracovisko 3 - Prekrocena teplota motora spodneho dopravnika !!!
    //A350 - Pracovisko 3 - Narusenie optickej bariery na vstupe !!!
    //A351 - Pracovisko 3 - Narusenie optickej bariery na vystupe !!!
    //A352 - Pracovisko 3 - Bolo stlacene tlacitko CS na rozvodnej skrini !!!
    //A353 - P3_Spodny stoper - Porucha vyvezenia paletky zo stopra !!!
    //A354 - P3_Vstupny stoper - Porucha vyvezenia paletky zo stopra !!!
    //A355 - ST7_Srobovanie - Porucha vyvezenia paletky zo stopra !!!
    //A356 - P3_Akumulacny stoper - Porucha vyvezenia paletky zo stopra !!!
    //A357 - ST8A_Leakage test A - Porucha vyvezenia paletky zo stopra !!!
    //A358 - ST8B_Leakage test B - Porucha vyvezenia paletky zo stopra !!!
    //A359 - ST7_Srobovanie - Porucha komunikacie s kamerou CAM 13 !!!
    //A360 - ST7_HV Test - Porucha vysunutia centrovacky !!!
	//A361 - ST7_HV Test - Porucha zasunutia centrovacky !!!
	//A362 - ST7_HV Test - Porucha vysunutia spodnych kontaktov !!!
	//A363 - ST7_HV Test - Porucha zasunutia spodnych kontaktov !!!
	//A364 - ST7_HV Test - Porucha vysunutia hornych kontaktov !!!
	//A365 - ST7_HV Test - Porucha zasunutia hornych kontaktov !!!
	//A366 - ST7_HV Test - Porucha precitania kodu paletky !!!
	//A367 - ST7_HV Test - Porucha vyvezenia paletky zo stopra !!!
	//A368 - P3_Zdvizka pred Leakage Testom A - Porucha vysunutia zdvizky !!!
	//A369 - P3_Zdvizka pred Leakage Testom A - Porucha zasunutia zdvizky !!!
	//A370 - P3_Zdvizka pred Leakage Testom A - Porucha strednej polohy zdvizky !!!
	//A371 - P3_Zdvizka pred Leakage Testom B - Porucha vysunutia zdvizky !!!
	//A372 - P3_Zdvizka pred Leakage Testom B - Porucha zasunutia zdvizky !!!
	//A373 - P3_Zdvizka pred Leakage Testom B - Porucha strednej polohy zdvizky !!!
	//A374 - P3_Zdvizka za Leakage Testom A - Porucha vysunutia zdvizky !!!
	//A375 - P3_Zdvizka za Leakage Testom A - Porucha zasunutia zdvizky !!!
	//A376 - P3_Zdvizka za Leakage Testom A - Porucha strednej polohy zdvizky !!!
	//A377 - P3_Zdvizka za Leakage Testom B - Porucha vysunutia zdvizky !!!
	//A378 - P3_Zdvizka za Leakage Testom B - Porucha zasunutia zdvizky !!!
	//A379 - P3_Zdvizka za Leakage Testom B - Porucha strednej polohy zdvizky !!!

	//Alarmy pracoviska č.4 (400 - 499)//
	//A400 - ST_Funkcny test A - porucha vysunutia centrovacky !!!
	//A401 - ST_Funkcny test A - porucha zasunutia centrovacky !!!
	//A402 - ST_Funkcny test B - porucha vysunutia centrovacky !!!
	//A403 - ST_Funkcny test B - porucha zasunutia centrovacky !!!
	//A404 - ST9_Etiketovacka - porucha vysunutia centrovacky !!!
	//A405 - ST9_Etiketovacka - porucha zasunutia centrovacky !!!
	//A406 - ST9_Etiketovacka - porucha precitania kodu paletky !!!
	//A407 - Pracovisko 4 - Porucha tlaku vzduchu !!!
	//A408 - ST9_Etiketovacka - porucha serva zdvihu aplikatora etikiet !!!
	//A409 - ST9_Etiketovacka - porucha komunikacie zo serverom !!!
	//A410 - ST10_Vytah - CAM 16 porucha komunikacie FTP !!!
	//A411 - ST10_Vytah - paletka na vystupe dopravnika vytahu !!!
	//A412 - ST10_Vytah - narusenie optickej bariery !!!
	//A413 - Pracovisko 4 - Kamera KAM15 a KAM16 nieje online !!!
	//A414 - Pracovisko 4 - Kamera KAM14 nieje online !!!
	//A415 - ST10_Vytah - porucha komunikacie zo serverom !!!
	//A416 - ST10_Vytah - porucha navezenia paletky na dopravnik vytahu !!!
	//A417 - Pracovisko 4 - Ventilovy termnal VT8 nieje online !!!
	//A418 - ST10_Vytah - porucha precitania kodu paletky !!!
	//A419 - ST_Funkcny test A - porucha vysunutia hornych kontaktov !!!
	//A420 - ST_Funkcny test A - porucha zasunutia hornych kontaktov !!!
	//A421 - ST_Funkcny test A - porucha vysunutia spodnych kontaktov !!!
	//A422 - ST_Funkcny test A - porucha zasunutia spodnych kontaktov !!!
	//A423 - ST_Funkcny test B - porucha vysunutia hornych kontaktov !!!
	//A424 - ST_Funkcny test B - porucha zasunutia hornych kontaktov !!!
	//A425 - ST_Funkcny test B - porucha vysunutia spodnych kontaktov !!!
	//A426 - ST_Funkcny test B - porucha zasunutia spodnych kontaktov !!!
	//A427 - ST_Funkcny test A - porucha precitania kodu paletky !!!
	//A428 - Pracovisko 4 - Modul DI41 nieje online !!!
	//A429 - ST_Funkcny test B - porucha precitania kodu paletky !!!
	//A430 - Pracovisko 4 - Modul DI42 nieje online !!!
	//A431 - ST9_Etiketovacka - porucha vytlacenie etikety !!!
	//A432 - ST9_Etiketovacka - pritlak pasky v tlaciarni je odisteny !!!
	//A433 - ST9_Etiketovacka - CAM 14 porucha komunikacie FTP !!!
	//A434 - ST9_Etiketovacka - CAM 15 porucha komunikacie FTP !!!
	//A435 - Pracovisko 4 - Modul DM41 nieje online !!!
	//A436 - Pracovisko 4 - Modul DS41 nieje online !!!
	//A437 - ST_Funkcny test A - je zalozeny nespravny typ spodneho kopita !!!
	//A438 - ST_Funkcny test B - je zalozeny nespravny typ spodneho kopita !!!
	//A439 - Pracovisko 4 - Modul DS42 nieje online !!!
    //A440 - Pracovisko 4 - Modul SI41 nieje online !!!
    //A441 - Pracovisko 4 - Modul SI42 nieje online !!!
    //A442 - ST10_Vytah - porucha serva zdvihu vytahu !!!
    //A443 - Pracovisko 4 - Prekrocena teplota motora vrchneho dopravnika !!!
    //A444 - Pracovisko 4 - Prekrocena teplota motora spodneho dopravnika !!!
    //A445 - ST10_Vytah - Prekrocena teplota motora dopravnika !!!
    //A446 - Pracovisko 4 - Narusenie optickej bariery na vstupe !!!
    //A447 - Pracovisko 4 - Narusenie optickej bariery na vystupe !!!
    //A448 - Pracovisko 4 - Bolo stlacene tlacitko CS na ovladacom paneli !!!
    //A449 - Pracovisko 4 - Bolo stlacene tlacitko CS na rozvodnej skrini !!!
    //A450 - ST_Funkcny test A - Porucha vyvezenia paletky zo stopra !!!
    //A451 - ST_Funkcny test B - Porucha vyvezenia paletky zo stopra !!!
    //A452 - ST9_Etiketovacka - Porucha vyvezenia paletky zo stopra !!!
    //A453 - ST9_Etiketovacka - Porucha komunikacie s kamerou CAM 14 !!!
    //A454 - ST9_Etiketovacka - Porucha komunikacie s kamerou CAM 15 !!!
    //A455 - ST10_Vytah - Porucha komunikacie s kamerou CAM 16 !!!
    //A456 - P4_Zdvizka za Funkcnym Testom A - Porucha vysunutia zdvizky !!!
	//A457 - P4_Zdvizka za Funkcnym Testom A - Porucha zasunutia zdvizky !!!
	//A458 - P4_Zdvizka za Funkcnym Testom A - Porucha strednej polohy zdvizky !!!
	//A459 - P4_Zdvizka za Funkcnym Testom B - Porucha vysunutia zdvizky !!!
	//A460 - P4_Zdvizka za Funkcnym Testom B - Porucha zasunutia zdvizky !!!
	//A461 - P4_Zdvizka za Funkcnym Testom B - Porucha strednej polohy zdvizky !!!
	//A462 - ST9_Etiketovacka - Porucha otocenia aplikatora vpred !!!
	//A463 - ST9_Etiketovacka - Porucha otocenia aplikatora vzad !!!

    //*********************Pracovisko 3 - Porucha tlaku vzduchu*********************************//
	IF CasKontroly_TlakVzduchuP3.Q THEN
		P34_Alarmy[323]:= TRUE;
		P3_Pracovisko.STAV.Porucha_ST1:= TRUE;
		P3_Pracovisko.STAV.Porucha_ST2:= TRUE;
		P3_Pracovisko.STAV.Porucha_ST3:= TRUE;
		P3_Pracovisko.STAV.Porucha_ST4:= TRUE;
		P3_Pracovisko.STAV.Porucha_ST5:= TRUE;
		P3_Pracovisko.STAV.Porucha_ST6:= TRUE;
		P3_Pracovisko.STAV.Porucha_ST7:= TRUE;
		P3_Pracovisko.STAV.Porucha_ST8:= TRUE;
	END_IF

	IF Safety.STAV.P3_ZonaBunky_AKTIVNA AND NOT P3_Pracovisko.IN.TlakVzduchu_OK THEN
		CasKontroly_TlakVzduchuP3.IN:= TRUE;
	ELSE
		CasKontroly_TlakVzduchuP3.IN:= FALSE;
	END_IF

	CasKontroly_TlakVzduchuP3.PT:= T#5s;
	CasKontroly_TlakVzduchuP3();

	//**********************************Porucha - IO moduly niesu online**************************************************//
	IF CasKontroly_ModulyP3.Q THEN
		P34_Alarmy[331]:= TRUE;
		P3_Pracovisko.STAV.Porucha_ST1:= TRUE;
		P3_Pracovisko.STAV.Porucha_ST2:= TRUE;
		P3_Pracovisko.STAV.Porucha_ST3:= TRUE;
		P3_Pracovisko.STAV.Porucha_ST4:= TRUE;
		P3_Pracovisko.STAV.Porucha_ST5:= TRUE;
		P3_Pracovisko.STAV.Porucha_ST6:= TRUE;
		P3_Pracovisko.STAV.Porucha_ST7:= TRUE;
		P3_Pracovisko.STAV.Porucha_ST8:= TRUE;
	END_IF

	IF Safety.STAV.P3_ZonaBunky_AKTIVNA AND (NOT P3_Pracovisko.IN.ModulFesto_IO_KomOK OR NOT P3_Pracovisko.IN.ModulWeidmuller_IO_KomOK) THEN
		CasKontroly_ModulyP3.IN:= TRUE;
	ELSE
		CasKontroly_ModulyP3.IN:= FALSE;
	END_IF

	CasKontroly_ModulyP3.PT:= T#2s;
	CasKontroly_ModulyP3();

	//********************************Porucha - ventilového terminálu**********************************************//
	IF CasKontroly_VentTerminalovP3.Q THEN
		P34_Alarmy[340]:= TRUE;
		P3_Pracovisko.STAV.Porucha_ST1:= TRUE;
		P3_Pracovisko.STAV.Porucha_ST2:= TRUE;
		P3_Pracovisko.STAV.Porucha_ST3:= TRUE;
		P3_Pracovisko.STAV.Porucha_ST4:= TRUE;
		P3_Pracovisko.STAV.Porucha_ST5:= TRUE;
		P3_Pracovisko.STAV.Porucha_ST6:= TRUE;
		P3_Pracovisko.STAV.Porucha_ST7:= TRUE;
		P3_Pracovisko.STAV.Porucha_ST8:= TRUE;
	END_IF

	IF Safety.STAV.P3_ZonaBunky_AKTIVNA AND NOT P3_Pracovisko.IN.VentilovyTerminal_KomOK THEN
		CasKontroly_VentTerminalovP3.IN:= TRUE;
	ELSE
		CasKontroly_VentTerminalovP3.IN:= FALSE;
	END_IF

	CasKontroly_VentTerminalovP3.PT:= T#2s;
	CasKontroly_VentTerminalovP3();

	//********************************Porucha - skrutkovacky niesu online**********************************************//
	IF CasKontroly_Skrutkovacky.Q THEN
		IF NOT P3_Pracovisko.IN.Skrutkovacka_K40_KomOK THEN
			P34_Alarmy[329]:= TRUE;
			P3_Pracovisko.STAV.Porucha_ST1:= TRUE;
		END_IF
		IF NOT P3_Pracovisko.IN.Skrutkovacka_M5_KomOK THEN
			P34_Alarmy[324]:= TRUE;
			P3_Pracovisko.STAV.Porucha_ST1:= TRUE;
		END_IF
	END_IF

	IF Safety.STAV.P3_ZonaBunky_AKTIVNA AND
		(NOT P3_Pracovisko.IN.Skrutkovacka_K40_KomOK OR
		NOT P3_Pracovisko.IN.Skrutkovacka_M5_KomOK) THEN
		CasKontroly_Skrutkovacky.IN:= TRUE;
	ELSE
		CasKontroly_Skrutkovacky.IN:= FALSE;
	END_IF

	CasKontroly_Skrutkovacky.PT:= T#2s;
	CasKontroly_Skrutkovacky();

	//*********************Pracovisko 3 - Porucha serva manipulatora šrobovania os Y***************//

	IF CasPoruchyServaSrobovaniaOsY.Q THEN
		P34_Alarmy[322]:= TRUE;
		P3_Pracovisko.STAV.Porucha_ST1:= TRUE;
	END_IF

	IF Safety.STAV.P3_ZonaBunky_AKTIVNA AND P3_Srobovanie.ServoManipulOsY.Status.Error THEN
		CasPoruchyServaSrobovaniaOsY.IN:= TRUE;
	ELSE
		CasPoruchyServaSrobovaniaOsY.IN:= FALSE;
	END_IF

	CasPoruchyServaSrobovaniaOsY.PT:= T#2s;
	CasPoruchyServaSrobovaniaOsY();

	//*********************Pracovisko 3 - Porucha serva manipulatora šrobovania os Z M5***************//
	IF CasPoruchyServaSrobovaniaOsZ_M5.Q THEN
		P34_Alarmy[332]:= TRUE;
		P3_Pracovisko.STAV.Porucha_ST1:= TRUE;
	END_IF

	IF Safety.STAV.P3_ZonaBunky_AKTIVNA AND P3_Srobovanie.ServoManipulOsZ_M5.Status.Error THEN
		CasPoruchyServaSrobovaniaOsZ_M5.IN:= TRUE;
	ELSE
		CasPoruchyServaSrobovaniaOsZ_M5.IN:= FALSE;
	END_IF

	CasPoruchyServaSrobovaniaOsZ_M5.PT:= T#2s;
	CasPoruchyServaSrobovaniaOsZ_M5();

	//********************Pracovisko 3 - Porucha skrutkovacieho setu M5******************************//
	IF P3_Srobovanie.Automat AND P3_Srobovanie.SkrutSet_M5.STAV.ERROR THEN
		P34_Alarmy[334]:= TRUE;
		P3_Pracovisko.STAV.Porucha_ST1:= TRUE;
	END_IF

	//****************************Pracovisko 3 - porucha predneho vrchného dopravníka**********************************//
	IF NOT P3_Dopravniky.IN.TeplotaMotoraPredDopravBunky_OK AND P3_Pracovisko.STAV.Automat THEN
		P34_Alarmy[348]:= TRUE;
		P3_Pracovisko.STAV.Porucha_ST1:= TRUE;
		P3_Pracovisko.STAV.Porucha_ST2:= TRUE;
		P3_Pracovisko.STAV.Porucha_ST3:= TRUE;
		P3_Pracovisko.STAV.Porucha_ST5:= TRUE;
		P3_Pracovisko.STAV.Porucha_ST7:= TRUE;
	END_IF

	//****************************Pracovisko 3 - porucha zadného vrchného dopravníka**********************************//
	IF NOT P3_Dopravniky.IN.TeplotaMotoraPredDopravBunky_OK AND P3_Pracovisko.STAV.Automat THEN
		P34_Alarmy[335]:= TRUE;
		P3_Pracovisko.STAV.Porucha_ST4:= TRUE;
		P3_Pracovisko.STAV.Porucha_ST6:= TRUE;
		P3_Pracovisko.STAV.Porucha_ST8:= TRUE;
	END_IF

	//*****************************Pracovisko 3 - porucha spodného dopravníka************************************//
	IF NOT P3_Dopravniky.IN.TeplotaMotoraVratnehoDoprav_OK AND P3_Pracovisko.STAV.Automat THEN
		P34_Alarmy[349]:= TRUE;
	END_IF

	//*****************************Pracovisko 3 - porucha prveho priecneho dopravníka************************************//
	IF NOT P3_Dopravniky.IN.TeplotaMotoraPriecnDoprav1_OK AND P3_Pracovisko.STAV.Automat THEN
		P34_Alarmy[336]:= TRUE;
	END_IF

	//*****************************Pracovisko 3 - porucha druheho priecneho dopravníka************************************//
	IF NOT P3_Dopravniky.IN.TeplotaMotoraPriecnDoprav2_OK AND P3_Pracovisko.STAV.Automat THEN
		P34_Alarmy[337]:= TRUE;
	END_IF

	//******************************Pracovisko 3 - narušenie vstupnej bariery bunky***********************************//
	IF NOT Safety.STAV.P3_Bunka_VstupBariera_AKTIVNA AND NOT Safety.STAV.P2_Bunka_Zamky_AKTIVNE AND NOT Safety.STAV.P2_VyblokovanieZamkov_AKTIVNE AND P3_Pracovisko.STAV.Automat THEN
		P34_Alarmy[350]:= TRUE;
		P3_Pracovisko.STAV.Porucha_ST1:= TRUE;
		P3_Pracovisko.STAV.Porucha_ST2:= TRUE;
		P3_Pracovisko.STAV.Porucha_ST3:= TRUE;
		P3_Pracovisko.STAV.Porucha_ST4:= TRUE;
		P3_Pracovisko.STAV.Porucha_ST5:= TRUE;
		P3_Pracovisko.STAV.Porucha_ST6:= TRUE;
		P3_Pracovisko.STAV.Porucha_ST7:= TRUE;
		P3_Pracovisko.STAV.Porucha_ST8:= TRUE;
	END_IF

	//******************************Pracovisko 3 - Stlačenie tlačítok CS*******************************************************//
	IF EDGENEG(Safety.STAV.P3_Rozvadzac_TlacitkoCS_ODBLOK) THEN
		P34_Alarmy[352]:= TRUE;
	END_IF

	//*********************Pracovisko 4 - Porucha tlaku vzduchu*********************************//
	IF CasKontroly_TlakVzduchuP4.Q THEN
		P34_Alarmy[407]:= TRUE;
		P4_Pracovisko.STAV.Porucha_ST1:= TRUE;
		P4_Pracovisko.STAV.Porucha_ST2:= TRUE;
		P4_Pracovisko.STAV.Porucha_ST3:= TRUE;
		P4_Pracovisko.STAV.Porucha_ST4:= TRUE;
		P4_Pracovisko.STAV.Porucha_ST5:= TRUE;
		P4_Pracovisko.STAV.Porucha_ST6:= TRUE;
	END_IF

	IF Safety.STAV.P4_ZonaBunky_AKTIVNA AND NOT P4_Pracovisko.IN.TlakVzduchu_OK THEN
		CasKontroly_TlakVzduchuP4.IN:= TRUE;
	ELSE
		CasKontroly_TlakVzduchuP4.IN:= FALSE;
	END_IF

	CasKontroly_TlakVzduchuP4.PT:= T#5s;
	CasKontroly_TlakVzduchuP4();

	//**********************************Porucha - kamerovy systém nieje online****************************************//
	IF CasKontroly_KAMsystemP4.Q THEN
		P34_Alarmy[413]:= TRUE;
		P4_Pracovisko.STAV.Porucha_ST5:= TRUE;
		P4_Pracovisko.STAV.Porucha_ST6:= TRUE;
	END_IF

	IF CasKontroly_KAM14.Q THEN
		P34_Alarmy[414]:= TRUE;
		P4_Pracovisko.STAV.Porucha_ST5:= TRUE;
	END_IF

	IF NOT P3_Pracovisko.IN.Kamery_ControlUnit_KomOK AND P4_Pracovisko.Automat THEN
		CasKontroly_KAMsystemP4.IN:= TRUE;
	ELSE
		CasKontroly_KAMsystemP4.IN:= FALSE;
	END_IF

	IF NOT CAM14.STAV.READY AND P4_Pracovisko.Automat THEN
		CasKontroly_KAM14.IN:= TRUE;
	ELSE
		CasKontroly_KAM14.IN:= FALSE;
	END_IF

	CasKontroly_KAMsystemP4.PT:= T#2s;
	CasKontroly_KAMsystemP4();
	CasKontroly_KAM14.PT:= T#2s;
	CasKontroly_KAM14();

	//**********************************Porucha - IO moduly niesu online**************************************************//
	IF CasKontroly_ModulyP4.Q THEN
		P34_Alarmy[428]:= TRUE;
		P4_Pracovisko.STAV.Porucha_ST1:= TRUE;
		P4_Pracovisko.STAV.Porucha_ST2:= TRUE;
		P4_Pracovisko.STAV.Porucha_ST3:= TRUE;
		P4_Pracovisko.STAV.Porucha_ST4:= TRUE;
		P4_Pracovisko.STAV.Porucha_ST5:= TRUE;
		P4_Pracovisko.STAV.Porucha_ST6:= TRUE;
	END_IF

	IF Safety.STAV.P4_ZonaBunky_AKTIVNA AND (NOT P4_Pracovisko.IN.ModulFesto_IO_KomOK OR NOT P4_Pracovisko.IN.ModulWeidmuller_IO_KomOK) THEN
		CasKontroly_ModulyP4.IN:= TRUE;
	ELSE
		CasKontroly_ModulyP4.IN:= FALSE;
	END_IF

	CasKontroly_ModulyP4.PT:= T#2s;
	CasKontroly_ModulyP4();

	//********************************Porucha - ventilového terminálu**********************************************//
	IF CasKontroly_VentTerminalovP4.Q THEN
		P34_Alarmy[417]:= TRUE;
		P4_Pracovisko.STAV.Porucha_ST1:= TRUE;
		P4_Pracovisko.STAV.Porucha_ST2:= TRUE;
		P4_Pracovisko.STAV.Porucha_ST3:= TRUE;
		P4_Pracovisko.STAV.Porucha_ST4:= TRUE;
		P4_Pracovisko.STAV.Porucha_ST5:= TRUE;
		P4_Pracovisko.STAV.Porucha_ST6:= TRUE;
	END_IF

	IF Safety.STAV.P4_ZonaBunky_AKTIVNA AND NOT P4_Pracovisko.IN.VentilovyTerminal_KomOK THEN
		CasKontroly_VentTerminalovP4.IN:= TRUE;
	ELSE
		CasKontroly_VentTerminalovP4.IN:= FALSE;
	END_IF

	CasKontroly_VentTerminalovP4.PT:= T#2s;
	CasKontroly_VentTerminalovP4();

	//*********************Pracovisko 4 - Porucha serva zdvihu aplikatora etikiet***************//

	IF CasPoruchyServaEtikety.Q THEN
		P34_Alarmy[408]:= TRUE;
		P4_Pracovisko.STAV.Porucha_ST5:= TRUE;
	END_IF

	IF Safety.STAV.P4_ZonaBunky_AKTIVNA AND P4_Etiketovacka.ServoZdvihuAplikatora.Status.Error THEN
		CasPoruchyServaEtikety.IN:= TRUE;
	ELSE
		CasPoruchyServaEtikety.IN:= FALSE;
	END_IF

	CasPoruchyServaEtikety.PT:= T#2s;
	CasPoruchyServaEtikety();

	//********************Pracovisko 4 - Porucha ochrannej bariéry výťahu****************************************//

	IF P4_Vytah.Automat AND NOT Safety.STAV.P4_Vytah_Bariera_AKTIVNA AND NOT Safety.STAV.P4_Vytah_Muting_AKTIVNY THEN
		P34_Alarmy[412]:= TRUE;
		P4_Pracovisko.STAV.Porucha_ST6:= TRUE;
	END_IF

	//*********************Pracovisko 4 - Porucha serva zdvihu vytahu***************//
	IF CasPoruchyServaVytahu.Q THEN
		P34_Alarmy[442]:= TRUE;
		P4_Pracovisko.STAV.Porucha_ST6:= TRUE;
	END_IF

	IF P4_Vytah.Automat AND P4_Vytah.ServoZdvihuVytahu.Status.Error THEN
		CasPoruchyServaVytahu.IN:= TRUE;
	ELSE
		CasPoruchyServaVytahu.IN:= FALSE;
	END_IF

	CasPoruchyServaVytahu.PT:= T#2s;
	CasPoruchyServaVytahu();

	//****************************Pracovisko 4 - porucha predneho vrchného dopravníka**********************************//
	IF NOT P4_Dopravniky.IN.TeplotaMotoraPredDopravBunky_OK AND P4_Pracovisko.STAV.Automat THEN
		P34_Alarmy[443]:= TRUE;
		P4_Pracovisko.STAV.Porucha_ST1:= TRUE;
		P4_Pracovisko.STAV.Porucha_ST3:= TRUE;
		P4_Pracovisko.STAV.Porucha_ST5:= TRUE;
	END_IF

	//****************************Pracovisko 4 - porucha zadneho vrchného dopravníka**********************************//
	IF NOT P4_Dopravniky.IN.TeplotaMotoraZadnDopravBunky_OK AND P4_Pracovisko.STAV.Automat THEN
		P34_Alarmy[430]:= TRUE;
		P4_Pracovisko.STAV.Porucha_ST2:= TRUE;
		P4_Pracovisko.STAV.Porucha_ST4:= TRUE;
	END_IF

	//*****************************Pracovisko 4 - porucha priecneho dopravníka************************************//
	IF NOT P4_Dopravniky.IN.TeplotaMotoraPriecnDoprav_OK AND P4_Pracovisko.STAV.Automat THEN
		P34_Alarmy[435]:= TRUE;
	END_IF

	//*****************************Pracovisko 4 - porucha spodného dopravníka************************************//
	IF NOT P4_Dopravniky.IN.TeplotaMotoraVratnehoDoprav_OK AND P4_Pracovisko.STAV.Automat THEN
		P34_Alarmy[444]:= TRUE;
	END_IF

	//******************************Pracovisko 4 - narušenie výstupnej bariery***********************************//

	IF CasKontrolyVystupnejBarieryP4.Q THEN
		P34_Alarmy[447]:= TRUE;
		P4_Pracovisko.STAV.Porucha_ST1:= TRUE;
		P4_Pracovisko.STAV.Porucha_ST2:= TRUE;
		P4_Pracovisko.STAV.Porucha_ST3:= TRUE;
		P4_Pracovisko.STAV.Porucha_ST4:= TRUE;
		P4_Pracovisko.STAV.Porucha_ST5:= TRUE;
	END_IF

	CasKontrolyVystupnejBarieryP4.IN:= NOT Safety.STAV.P4_VystupBunky_VstupBar_AKTIVNA AND NOT Safety.STAV.P4_VystupBunky_VystupBar_AKTIVNA AND P4_Pracovisko.STAV.Automat;
	CasKontrolyVystupnejBarieryP4.PT:= T#500ms;
	CasKontrolyVystupnejBarieryP4();

	//******************************Výťah - porucha dopravníka**************************************************//
	IF NOT P4_Vytah.IN.TeplotaMotoraDopravVytahu_OK AND P4_Vytah.Automat THEN
		P34_Alarmy[445]:= TRUE;
		P4_Pracovisko.STAV.Porucha_ST6:= TRUE;
	END_IF

	//******************************Pracovisko 4 - Stlačenie tlačítok CS*******************************************************//
	IF EDGENEG(Safety.STAV.P4_Panel_TlacitkoCS_ODBLOK) THEN
		P34_Alarmy[448]:= TRUE;
	END_IF

	IF EDGENEG(Safety.STAV.P4_Rozvadzac_TlacitkoCS_ODBLOK) THEN
		P34_Alarmy[449]:= TRUE;
	END_IF

	//***************************************************Nasetovanie alarmov****************************************************//
	//Pracovisko č.3//
	IF P34_Alarmy[300] THEN
		MpAlarmXSet(gAlarmXCore, 'A300');
	ELSE
		MpAlarmXReset(gAlarmXCore, 'A300');
	END_IF

	IF P34_Alarmy[301] THEN
		MpAlarmXSet(gAlarmXCore, 'A301');
	ELSE
		MpAlarmXReset(gAlarmXCore, 'A301');
	END_IF

	IF P34_Alarmy[302] THEN
		MpAlarmXSet(gAlarmXCore, 'A302');
	ELSE
		MpAlarmXReset(gAlarmXCore, 'A302');
	END_IF

	IF P34_Alarmy[303] THEN
		MpAlarmXSet(gAlarmXCore, 'A303');
	ELSE
		MpAlarmXReset(gAlarmXCore, 'A303');
	END_IF

	IF P34_Alarmy[304] THEN
		MpAlarmXSet(gAlarmXCore, 'A304');
	ELSE
		MpAlarmXReset(gAlarmXCore, 'A304');
	END_IF

	IF P34_Alarmy[305] THEN
		MpAlarmXSet(gAlarmXCore, 'A305');
	ELSE
		MpAlarmXReset(gAlarmXCore, 'A305');
	END_IF

	IF P34_Alarmy[306] THEN
		MpAlarmXSet(gAlarmXCore, 'A306');
	ELSE
		MpAlarmXReset(gAlarmXCore, 'A306');
	END_IF

	IF P34_Alarmy[307] THEN
		MpAlarmXSet(gAlarmXCore, 'A307');
	ELSE
		MpAlarmXReset(gAlarmXCore, 'A307');
	END_IF

	IF P34_Alarmy[308] THEN
		MpAlarmXSet(gAlarmXCore, 'A308');
	ELSE
		MpAlarmXReset(gAlarmXCore, 'A308');
	END_IF

	IF P34_Alarmy[309] THEN
		MpAlarmXSet(gAlarmXCore, 'A309');
	ELSE
		MpAlarmXReset(gAlarmXCore, 'A309');
	END_IF

	IF P34_Alarmy[310] THEN
		MpAlarmXSet(gAlarmXCore, 'A310');
	ELSE
		MpAlarmXReset(gAlarmXCore, 'A310');
	END_IF

	IF P34_Alarmy[311] THEN
		MpAlarmXSet(gAlarmXCore, 'A311');
	ELSE
		MpAlarmXReset(gAlarmXCore, 'A311');
	END_IF

	IF P34_Alarmy[312] THEN
		MpAlarmXSet(gAlarmXCore, 'A312');
	ELSE
		MpAlarmXReset(gAlarmXCore, 'A312');
	END_IF

	IF P34_Alarmy[313] THEN
		MpAlarmXSet(gAlarmXCore, 'A313');
	ELSE
		MpAlarmXReset(gAlarmXCore, 'A313');
	END_IF

	IF P34_Alarmy[314] THEN
		MpAlarmXSet(gAlarmXCore, 'A314');
	ELSE
		MpAlarmXReset(gAlarmXCore, 'A314');
	END_IF

	IF P34_Alarmy[315] THEN
		MpAlarmXSet(gAlarmXCore, 'A315');
	ELSE
		MpAlarmXReset(gAlarmXCore, 'A315');
	END_IF

	IF P34_Alarmy[316] THEN
		MpAlarmXSet(gAlarmXCore, 'A316');
	ELSE
		MpAlarmXReset(gAlarmXCore, 'A316');
	END_IF

	IF P34_Alarmy[317] THEN
		MpAlarmXSet(gAlarmXCore, 'A317');
	ELSE
		MpAlarmXReset(gAlarmXCore, 'A317');
	END_IF

	IF P34_Alarmy[318] THEN
		MpAlarmXSet(gAlarmXCore, 'A318');
	ELSE
		MpAlarmXReset(gAlarmXCore, 'A318');
	END_IF

	IF P34_Alarmy[319] THEN
		MpAlarmXSet(gAlarmXCore, 'A319');
	ELSE
		MpAlarmXReset(gAlarmXCore, 'A319');
	END_IF

	IF P34_Alarmy[320] THEN
		MpAlarmXSet(gAlarmXCore, 'A320');
	ELSE
		MpAlarmXReset(gAlarmXCore, 'A320');
	END_IF

	IF P34_Alarmy[321] THEN
		MpAlarmXSet(gAlarmXCore, 'A321');
	ELSE
		MpAlarmXReset(gAlarmXCore, 'A321');
	END_IF

	IF P34_Alarmy[322] THEN
		MpAlarmXSet(gAlarmXCore, 'A322');
	ELSE
		MpAlarmXReset(gAlarmXCore, 'A322');
	END_IF

	IF P34_Alarmy[323] THEN
		MpAlarmXSet(gAlarmXCore, 'A323');
	ELSE
		MpAlarmXReset(gAlarmXCore, 'A323');
	END_IF

	IF P34_Alarmy[324] THEN
		MpAlarmXSet(gAlarmXCore, 'A324');
	ELSE
		MpAlarmXReset(gAlarmXCore, 'A324');
	END_IF

	IF P34_Alarmy[325] THEN
		MpAlarmXSet(gAlarmXCore, 'A325');
	ELSE
		MpAlarmXReset(gAlarmXCore, 'A325');
	END_IF

	IF P34_Alarmy[326] THEN
		MpAlarmXSet(gAlarmXCore, 'A326');
	ELSE
		MpAlarmXReset(gAlarmXCore, 'A326');
	END_IF

	IF P34_Alarmy[327] THEN
		MpAlarmXSet(gAlarmXCore, 'A327');
	ELSE
		MpAlarmXReset(gAlarmXCore, 'A327');
	END_IF

	IF P34_Alarmy[328] THEN
		MpAlarmXSet(gAlarmXCore, 'A328');
	ELSE
		MpAlarmXReset(gAlarmXCore, 'A328');
	END_IF

	IF P34_Alarmy[329] THEN
		MpAlarmXSet(gAlarmXCore, 'A329');
	ELSE
		MpAlarmXReset(gAlarmXCore, 'A329');
	END_IF

	IF P34_Alarmy[330] THEN
		MpAlarmXSet(gAlarmXCore, 'A330');
	ELSE
		MpAlarmXReset(gAlarmXCore, 'A330');
	END_IF

	IF P34_Alarmy[331] THEN
		MpAlarmXSet(gAlarmXCore, 'A331');
	ELSE
		MpAlarmXReset(gAlarmXCore, 'A331');
	END_IF

	IF P34_Alarmy[332] THEN
		MpAlarmXSet(gAlarmXCore, 'A332');
	ELSE
		MpAlarmXReset(gAlarmXCore, 'A332');
	END_IF

	IF P34_Alarmy[333] THEN
		MpAlarmXSet(gAlarmXCore, 'A333');
	ELSE
		MpAlarmXReset(gAlarmXCore, 'A333');
	END_IF

	IF P34_Alarmy[334] THEN
		MpAlarmXSet(gAlarmXCore, 'A334');
	ELSE
		MpAlarmXReset(gAlarmXCore, 'A334');
	END_IF

	IF P34_Alarmy[335] THEN
		MpAlarmXSet(gAlarmXCore, 'A335');
	ELSE
		MpAlarmXReset(gAlarmXCore, 'A335');
	END_IF

	IF P34_Alarmy[336] THEN
		MpAlarmXSet(gAlarmXCore, 'A336');
	ELSE
		MpAlarmXReset(gAlarmXCore, 'A336');
	END_IF

	IF P34_Alarmy[337] THEN
		MpAlarmXSet(gAlarmXCore, 'A337');
	ELSE
		MpAlarmXReset(gAlarmXCore, 'A337');
	END_IF

	IF P34_Alarmy[338] THEN
		MpAlarmXSet(gAlarmXCore, 'A338');
	ELSE
		MpAlarmXReset(gAlarmXCore, 'A338');
	END_IF

	IF P34_Alarmy[339] THEN
		MpAlarmXSet(gAlarmXCore, 'A339');
	ELSE
		MpAlarmXReset(gAlarmXCore, 'A339');
	END_IF

	IF P34_Alarmy[340] THEN
		MpAlarmXSet(gAlarmXCore, 'A340');
	ELSE
		MpAlarmXReset(gAlarmXCore, 'A340');
	END_IF

	IF P34_Alarmy[341] THEN
		MpAlarmXSet(gAlarmXCore, 'A341');
	ELSE
		MpAlarmXReset(gAlarmXCore, 'A341');
	END_IF

	IF P34_Alarmy[342] THEN
		MpAlarmXSet(gAlarmXCore, 'A342');
	ELSE
		MpAlarmXReset(gAlarmXCore, 'A342');
	END_IF

	IF P34_Alarmy[343] THEN
		MpAlarmXSet(gAlarmXCore, 'A343');
	ELSE
		MpAlarmXReset(gAlarmXCore, 'A343');
	END_IF

	IF P34_Alarmy[344] THEN
		MpAlarmXSet(gAlarmXCore, 'A344');
	ELSE
		MpAlarmXReset(gAlarmXCore, 'A344');
	END_IF

	IF P34_Alarmy[345] THEN
		MpAlarmXSet(gAlarmXCore, 'A345');
	ELSE
		MpAlarmXReset(gAlarmXCore, 'A345');
	END_IF

	IF P34_Alarmy[346] THEN
		MpAlarmXSet(gAlarmXCore, 'A346');
	ELSE
		MpAlarmXReset(gAlarmXCore, 'A346');
	END_IF

	IF P34_Alarmy[347] THEN
		MpAlarmXSet(gAlarmXCore, 'A347');
	ELSE
		MpAlarmXReset(gAlarmXCore, 'A347');
	END_IF

	IF P34_Alarmy[348] THEN
		MpAlarmXSet(gAlarmXCore, 'A348');
	ELSE
		MpAlarmXReset(gAlarmXCore, 'A348');
	END_IF

	IF P34_Alarmy[349] THEN
		MpAlarmXSet(gAlarmXCore, 'A349');
	ELSE
		MpAlarmXReset(gAlarmXCore, 'A349');
	END_IF

	IF P34_Alarmy[350] THEN
		MpAlarmXSet(gAlarmXCore, 'A350');
	ELSE
		MpAlarmXReset(gAlarmXCore, 'A350');
	END_IF

	IF P34_Alarmy[351] THEN
		MpAlarmXSet(gAlarmXCore, 'A351');
	ELSE
		MpAlarmXReset(gAlarmXCore, 'A351');
	END_IF

	IF P34_Alarmy[352] THEN
		MpAlarmXSet(gAlarmXCore, 'A352');
	ELSE
		MpAlarmXReset(gAlarmXCore, 'A352');
	END_IF

	IF P34_Alarmy[353] THEN
		MpAlarmXSet(gAlarmXCore, 'A353');
	ELSE
		MpAlarmXReset(gAlarmXCore, 'A353');
	END_IF

	IF P34_Alarmy[354] THEN
		MpAlarmXSet(gAlarmXCore, 'A354');
	ELSE
		MpAlarmXReset(gAlarmXCore, 'A354');
	END_IF

	IF P34_Alarmy[355] THEN
		MpAlarmXSet(gAlarmXCore, 'A355');
	ELSE
		MpAlarmXReset(gAlarmXCore, 'A355');
	END_IF

	IF P34_Alarmy[356] THEN
		MpAlarmXSet(gAlarmXCore, 'A356');
	ELSE
		MpAlarmXReset(gAlarmXCore, 'A356');
	END_IF

	IF P34_Alarmy[357] THEN
		MpAlarmXSet(gAlarmXCore, 'A357');
	ELSE
		MpAlarmXReset(gAlarmXCore, 'A357');
	END_IF

	IF P34_Alarmy[358] THEN
		MpAlarmXSet(gAlarmXCore, 'A358');
	ELSE
		MpAlarmXReset(gAlarmXCore, 'A358');
	END_IF

	IF P34_Alarmy[359] THEN
		MpAlarmXSet(gAlarmXCore, 'A359');
	ELSE
		MpAlarmXReset(gAlarmXCore, 'A359');
	END_IF

	IF P34_Alarmy[360] THEN
		MpAlarmXSet(gAlarmXCore, 'A360');
	ELSE
		MpAlarmXReset(gAlarmXCore, 'A360');
	END_IF

	IF P34_Alarmy[361] THEN
		MpAlarmXSet(gAlarmXCore, 'A362');
	ELSE
		MpAlarmXReset(gAlarmXCore, 'A362');
	END_IF

	IF P34_Alarmy[362] THEN
		MpAlarmXSet(gAlarmXCore, 'A362');
	ELSE
		MpAlarmXReset(gAlarmXCore, 'A362');
	END_IF

	IF P34_Alarmy[363] THEN
		MpAlarmXSet(gAlarmXCore, 'A363');
	ELSE
		MpAlarmXReset(gAlarmXCore, 'A363');
	END_IF

	IF P34_Alarmy[364] THEN
		MpAlarmXSet(gAlarmXCore, 'A364');
	ELSE
		MpAlarmXReset(gAlarmXCore, 'A364');
	END_IF

	IF P34_Alarmy[365] THEN
		MpAlarmXSet(gAlarmXCore, 'A365');
	ELSE
		MpAlarmXReset(gAlarmXCore, 'A365');
	END_IF

	IF P34_Alarmy[366] THEN
		MpAlarmXSet(gAlarmXCore, 'A366');
	ELSE
		MpAlarmXReset(gAlarmXCore, 'A366');
	END_IF

	IF P34_Alarmy[367] THEN
		MpAlarmXSet(gAlarmXCore, 'A367');
	ELSE
		MpAlarmXReset(gAlarmXCore, 'A367');
	END_IF

	IF P34_Alarmy[368] THEN
		MpAlarmXSet(gAlarmXCore, 'A368');
	ELSE
		MpAlarmXReset(gAlarmXCore, 'A368');
	END_IF

	IF P34_Alarmy[369] THEN
		MpAlarmXSet(gAlarmXCore, 'A369');
	ELSE
		MpAlarmXReset(gAlarmXCore, 'A369');
	END_IF

	IF P34_Alarmy[370] THEN
		MpAlarmXSet(gAlarmXCore, 'A370');
	ELSE
		MpAlarmXReset(gAlarmXCore, 'A370');
	END_IF

	IF P34_Alarmy[371] THEN
		MpAlarmXSet(gAlarmXCore, 'A371');
	ELSE
		MpAlarmXReset(gAlarmXCore, 'A371');
	END_IF

	IF P34_Alarmy[372] THEN
		MpAlarmXSet(gAlarmXCore, 'A372');
	ELSE
		MpAlarmXReset(gAlarmXCore, 'A372');
	END_IF

	IF P34_Alarmy[373] THEN
		MpAlarmXSet(gAlarmXCore, 'A373');
	ELSE
		MpAlarmXReset(gAlarmXCore, 'A373');
	END_IF

	IF P34_Alarmy[374] THEN
		MpAlarmXSet(gAlarmXCore, 'A374');
	ELSE
		MpAlarmXReset(gAlarmXCore, 'A374');
	END_IF

	IF P34_Alarmy[375] THEN
		MpAlarmXSet(gAlarmXCore, 'A375');
	ELSE
		MpAlarmXReset(gAlarmXCore, 'A375');
	END_IF

	IF P34_Alarmy[376] THEN
		MpAlarmXSet(gAlarmXCore, 'A376');
	ELSE
		MpAlarmXReset(gAlarmXCore, 'A376');
	END_IF

	IF P34_Alarmy[377] THEN
		MpAlarmXSet(gAlarmXCore, 'A377');
	ELSE
		MpAlarmXReset(gAlarmXCore, 'A377');
	END_IF

	IF P34_Alarmy[378] THEN
		MpAlarmXSet(gAlarmXCore, 'A378');
	ELSE
		MpAlarmXReset(gAlarmXCore, 'A378');
	END_IF

	IF P34_Alarmy[379] THEN
		MpAlarmXSet(gAlarmXCore, 'A379');
	ELSE
		MpAlarmXReset(gAlarmXCore, 'A379');
	END_IF

	//Pracovisko č.4//

	IF P34_Alarmy[400] THEN
		MpAlarmXSet(gAlarmXCore, 'A400');
	ELSE
		MpAlarmXReset(gAlarmXCore, 'A400');
	END_IF

	IF P34_Alarmy[401] THEN
		MpAlarmXSet(gAlarmXCore, 'A401');
	ELSE
		MpAlarmXReset(gAlarmXCore, 'A401');
	END_IF

	IF P34_Alarmy[402] THEN
		MpAlarmXSet(gAlarmXCore, 'A402');
	ELSE
		MpAlarmXReset(gAlarmXCore, 'A402');
	END_IF

	IF P34_Alarmy[403] THEN
		MpAlarmXSet(gAlarmXCore, 'A403');
	ELSE
		MpAlarmXReset(gAlarmXCore, 'A403');
	END_IF

	IF P34_Alarmy[404] THEN
		MpAlarmXSet(gAlarmXCore, 'A404');
	ELSE
		MpAlarmXReset(gAlarmXCore, 'A404');
	END_IF

	IF P34_Alarmy[405] THEN
		MpAlarmXSet(gAlarmXCore, 'A405');
	ELSE
		MpAlarmXReset(gAlarmXCore, 'A405');
	END_IF

	IF P34_Alarmy[406] THEN
		MpAlarmXSet(gAlarmXCore, 'A406');
	ELSE
		MpAlarmXReset(gAlarmXCore, 'A406');
	END_IF

	IF P34_Alarmy[407] THEN
		MpAlarmXSet(gAlarmXCore, 'A407');
	ELSE
		MpAlarmXReset(gAlarmXCore, 'A407');
	END_IF

	IF P34_Alarmy[408] THEN
		MpAlarmXSet(gAlarmXCore, 'A408');
	ELSE
		MpAlarmXReset(gAlarmXCore, 'A408');
	END_IF

	IF P34_Alarmy[409] THEN
		MpAlarmXSet(gAlarmXCore, 'A409');
	ELSE
		MpAlarmXReset(gAlarmXCore, 'A409');
	END_IF

	IF P34_Alarmy[410] THEN
		MpAlarmXSet(gAlarmXCore, 'A410');
	ELSE
		MpAlarmXReset(gAlarmXCore, 'A410');
	END_IF

	IF P34_Alarmy[411] THEN
		MpAlarmXSet(gAlarmXCore, 'A411');
	ELSE
		MpAlarmXReset(gAlarmXCore, 'A411');
	END_IF

	IF P34_Alarmy[412] THEN
		MpAlarmXSet(gAlarmXCore, 'A412');
	ELSE
		MpAlarmXReset(gAlarmXCore, 'A412');
	END_IF

	IF P34_Alarmy[413] THEN
		MpAlarmXSet(gAlarmXCore, 'A413');
	ELSE
		MpAlarmXReset(gAlarmXCore, 'A413');
	END_IF

	IF P34_Alarmy[414] THEN
		MpAlarmXSet(gAlarmXCore, 'A414');
	ELSE
		MpAlarmXReset(gAlarmXCore, 'A414');
	END_IF

	IF P34_Alarmy[415] THEN
		MpAlarmXSet(gAlarmXCore, 'A415');
	ELSE
		MpAlarmXReset(gAlarmXCore, 'A415');
	END_IF

	IF P34_Alarmy[416] THEN
		MpAlarmXSet(gAlarmXCore, 'A416');
	ELSE
		MpAlarmXReset(gAlarmXCore, 'A416');
	END_IF

	IF P34_Alarmy[417] THEN
		MpAlarmXSet(gAlarmXCore, 'A417');
	ELSE
		MpAlarmXReset(gAlarmXCore, 'A417');
	END_IF

	IF P34_Alarmy[418] THEN
		MpAlarmXSet(gAlarmXCore, 'A418');
	ELSE
		MpAlarmXReset(gAlarmXCore, 'A418');
	END_IF

	IF P34_Alarmy[419] THEN
		MpAlarmXSet(gAlarmXCore, 'A419');
	ELSE
		MpAlarmXReset(gAlarmXCore, 'A419');
	END_IF

	IF P34_Alarmy[420] THEN
		MpAlarmXSet(gAlarmXCore, 'A420');
	ELSE
		MpAlarmXReset(gAlarmXCore, 'A420');
	END_IF

	IF P34_Alarmy[421] THEN
		MpAlarmXSet(gAlarmXCore, 'A421');
	ELSE
		MpAlarmXReset(gAlarmXCore, 'A421');
	END_IF

	IF P34_Alarmy[422] THEN
		MpAlarmXSet(gAlarmXCore, 'A422');
	ELSE
		MpAlarmXReset(gAlarmXCore, 'A422');
	END_IF

	IF P34_Alarmy[423] THEN
		MpAlarmXSet(gAlarmXCore, 'A423');
	ELSE
		MpAlarmXReset(gAlarmXCore, 'A423');
	END_IF

	IF P34_Alarmy[424] THEN
		MpAlarmXSet(gAlarmXCore, 'A424');
	ELSE
		MpAlarmXReset(gAlarmXCore, 'A424');
	END_IF

	IF P34_Alarmy[425] THEN
		MpAlarmXSet(gAlarmXCore, 'A425');
	ELSE
		MpAlarmXReset(gAlarmXCore, 'A425');
	END_IF

	IF P34_Alarmy[426] THEN
		MpAlarmXSet(gAlarmXCore, 'A426');
	ELSE
		MpAlarmXReset(gAlarmXCore, 'A426');
	END_IF

	IF P34_Alarmy[427] THEN
		MpAlarmXSet(gAlarmXCore, 'A427');
	ELSE
		MpAlarmXReset(gAlarmXCore, 'A427');
	END_IF

	IF P34_Alarmy[428] THEN
		MpAlarmXSet(gAlarmXCore, 'A428');
	ELSE
		MpAlarmXReset(gAlarmXCore, 'A428');
	END_IF

	IF P34_Alarmy[429] THEN
		MpAlarmXSet(gAlarmXCore, 'A429');
	ELSE
		MpAlarmXReset(gAlarmXCore, 'A429');
	END_IF

	IF P34_Alarmy[430] THEN
		MpAlarmXSet(gAlarmXCore, 'A430');
	ELSE
		MpAlarmXReset(gAlarmXCore, 'A430');
	END_IF

	IF P34_Alarmy[431] THEN
		MpAlarmXSet(gAlarmXCore, 'A431');
	ELSE
		MpAlarmXReset(gAlarmXCore, 'A431');
	END_IF

	IF P34_Alarmy[432] THEN
		MpAlarmXSet(gAlarmXCore, 'A432');
	ELSE
		MpAlarmXReset(gAlarmXCore, 'A432');
	END_IF

	IF P34_Alarmy[433] THEN
		MpAlarmXSet(gAlarmXCore, 'A433');
	ELSE
		MpAlarmXReset(gAlarmXCore, 'A433');
	END_IF

	IF P34_Alarmy[434] THEN
		MpAlarmXSet(gAlarmXCore, 'A434');
	ELSE
		MpAlarmXReset(gAlarmXCore, 'A434');
	END_IF

	IF P34_Alarmy[435] THEN
		MpAlarmXSet(gAlarmXCore, 'A435');
	ELSE
		MpAlarmXReset(gAlarmXCore, 'A435');
	END_IF

	IF P34_Alarmy[436] THEN
		MpAlarmXSet(gAlarmXCore, 'A436');
	ELSE
		MpAlarmXReset(gAlarmXCore, 'A436');
	END_IF

	IF P34_Alarmy[437] THEN
		MpAlarmXSet(gAlarmXCore, 'A437');
	ELSE
		MpAlarmXReset(gAlarmXCore, 'A437');
	END_IF

	IF P34_Alarmy[438] THEN
		MpAlarmXSet(gAlarmXCore, 'A438');
	ELSE
		MpAlarmXReset(gAlarmXCore, 'A438');
	END_IF

	IF P34_Alarmy[439] THEN
		MpAlarmXSet(gAlarmXCore, 'A439');
	ELSE
		MpAlarmXReset(gAlarmXCore, 'A439');
	END_IF

	IF P34_Alarmy[440] THEN
		MpAlarmXSet(gAlarmXCore, 'A440');
	ELSE
		MpAlarmXReset(gAlarmXCore, 'A440');
	END_IF

	IF P34_Alarmy[441] THEN
		MpAlarmXSet(gAlarmXCore, 'A441');
	ELSE
		MpAlarmXReset(gAlarmXCore, 'A441');
	END_IF

	IF P34_Alarmy[442] THEN
		MpAlarmXSet(gAlarmXCore, 'A442');
	ELSE
		MpAlarmXReset(gAlarmXCore, 'A442');
	END_IF

	IF P34_Alarmy[443] THEN
		MpAlarmXSet(gAlarmXCore, 'A443');
	ELSE
		MpAlarmXReset(gAlarmXCore, 'A443');
	END_IF

	IF P34_Alarmy[444] THEN
		MpAlarmXSet(gAlarmXCore, 'A444');
	ELSE
		MpAlarmXReset(gAlarmXCore, 'A444');
	END_IF

	IF P34_Alarmy[445] THEN
		MpAlarmXSet(gAlarmXCore, 'A445');
	ELSE
		MpAlarmXReset(gAlarmXCore, 'A445');
	END_IF

	IF P34_Alarmy[446] THEN
		MpAlarmXSet(gAlarmXCore, 'A446');
	ELSE
		MpAlarmXReset(gAlarmXCore, 'A446');
	END_IF

	IF P34_Alarmy[447] THEN
		MpAlarmXSet(gAlarmXCore, 'A447');
	ELSE
		MpAlarmXReset(gAlarmXCore, 'A447');
	END_IF

	IF P34_Alarmy[448] THEN
		MpAlarmXSet(gAlarmXCore, 'A448');
	ELSE
		MpAlarmXReset(gAlarmXCore, 'A448');
	END_IF

	IF P34_Alarmy[449] THEN
		MpAlarmXSet(gAlarmXCore, 'A449');
	ELSE
		MpAlarmXReset(gAlarmXCore, 'A449');
	END_IF

	IF P34_Alarmy[450] THEN
		MpAlarmXSet(gAlarmXCore, 'A450');
	ELSE
		MpAlarmXReset(gAlarmXCore, 'A450');
	END_IF

	IF P34_Alarmy[451] THEN
		MpAlarmXSet(gAlarmXCore, 'A451');
	ELSE
		MpAlarmXReset(gAlarmXCore, 'A451');
	END_IF

	IF P34_Alarmy[452] THEN
		MpAlarmXSet(gAlarmXCore, 'A452');
	ELSE
		MpAlarmXReset(gAlarmXCore, 'A452');
	END_IF

	IF P34_Alarmy[453] THEN
		MpAlarmXSet(gAlarmXCore, 'A453');
	ELSE
		MpAlarmXReset(gAlarmXCore, 'A453');
	END_IF

	IF P34_Alarmy[454] THEN
		MpAlarmXSet(gAlarmXCore, 'A454');
	ELSE
		MpAlarmXReset(gAlarmXCore, 'A454');
	END_IF

	IF P34_Alarmy[455] THEN
		MpAlarmXSet(gAlarmXCore, 'A455');
	ELSE
		MpAlarmXReset(gAlarmXCore, 'A455');
	END_IF

	IF P34_Alarmy[456] THEN
		MpAlarmXSet(gAlarmXCore, 'A456');
	ELSE
		MpAlarmXReset(gAlarmXCore, 'A456');
	END_IF

	IF P34_Alarmy[457] THEN
		MpAlarmXSet(gAlarmXCore, 'A457');
	ELSE
		MpAlarmXReset(gAlarmXCore, 'A457');
	END_IF

	IF P34_Alarmy[458] THEN
		MpAlarmXSet(gAlarmXCore, 'A458');
	ELSE
		MpAlarmXReset(gAlarmXCore, 'A458');
	END_IF

	IF P34_Alarmy[459] THEN
		MpAlarmXSet(gAlarmXCore, 'A459');
	ELSE
		MpAlarmXReset(gAlarmXCore, 'A459');
	END_IF

	IF P34_Alarmy[460] THEN
		MpAlarmXSet(gAlarmXCore, 'A460');
	ELSE
		MpAlarmXReset(gAlarmXCore, 'A460');
	END_IF

	IF P34_Alarmy[461] THEN
		MpAlarmXSet(gAlarmXCore, 'A461');
	ELSE
		MpAlarmXReset(gAlarmXCore, 'A461');
	END_IF

	IF P34_Alarmy[462] THEN
		MpAlarmXSet(gAlarmXCore, 'A462');
	ELSE
		MpAlarmXReset(gAlarmXCore, 'A462');
	END_IF

	IF P34_Alarmy[463] THEN
		MpAlarmXSet(gAlarmXCore, 'A463');
	ELSE
		MpAlarmXReset(gAlarmXCore, 'A463');
	END_IF

	//*************************************Potvrdenie alarmov*********************************************************//
	IF P34_AlarmyVizu.PotvrdAlarmy THEN
		brsmemset(ADR(P34_Alarmy),0,SIZEOF(P34_Alarmy));
		P3_Pracovisko.STAV.Porucha_ST1:= FALSE;
		P3_Pracovisko.STAV.Porucha_ST2:= FALSE;
		P3_Pracovisko.STAV.Porucha_ST3:= FALSE;
		P3_Pracovisko.STAV.Porucha_ST4:= FALSE;
		P3_Pracovisko.STAV.Porucha_ST5:= FALSE;
		P3_Pracovisko.STAV.Porucha_ST6:= FALSE;
		P3_Pracovisko.STAV.Porucha_ST7:= FALSE;
		P3_Pracovisko.STAV.Porucha_ST8:= FALSE;
		P4_Pracovisko.STAV.Porucha_ST1:= FALSE;
		P4_Pracovisko.STAV.Porucha_ST2:= FALSE;
		P4_Pracovisko.STAV.Porucha_ST3:= FALSE;
		P4_Pracovisko.STAV.Porucha_ST4:= FALSE;
		P4_Pracovisko.STAV.Porucha_ST5:= FALSE;
		P4_Pracovisko.STAV.Porucha_ST6:= FALSE;
		IF NOT P4_Vytah.Automat THEN
			P4_Vytah.ServoZdvihuVytahu.Command.ErrReset:= TRUE;
		END_IF
		IF NOT P3_Srobovanie.Automat THEN
			P3_Srobovanie.ServoManipulOsY.Command.ErrReset:= TRUE;
			P3_Srobovanie.SkrutSet_M5.CMD.ResetPoruchy:= TRUE;
		END_IF
		IF NOT P4_Etiketovacka.Automat THEN
			P4_Etiketovacka.ServoZdvihuAplikatora.Command.ErrReset:= TRUE;
		END_IF
		P34_AlarmyVizu.PotvrdAlarmy:= FALSE;
	END_IF

        END_PROGRAM

PROGRAM _EXIT
        (* Insert code here *)

        END_PROGRAM
```

#### Variables.var - Local variables
```iecst
VAR
	i : UINT;
	CasKontroly_TlakVzduchuP3 : TON;
	CasKontroly_KAMsystemP3 : TON;
	CasKontroly_ModulyP3 : TON;
	CasKontroly_VentTerminalovP3 : TON;
	CasKontroly_Skrutkovacky : TON;
	CasKontroly_TlakVzduchuP4 : TON;
	CasKontroly_KAMsystemP4 : TON;
	CasKontroly_ModulyP4 : TON;
	CasKontroly_VentTerminalovP4 : TON;
	CasPoruchyServaVytahu : TON;
	CasPoruchyServaSrobovaniaOsY : TON;
	CasPoruchyServaEtikety : TON;
	CasResetovaniaServaZdvihuVytahu : TON;
	CasResetServaZdvihuEtiketovacky : TON;
	CasResetovaniaServaSrobovaniaOsY : TON;
	a : INT;
	b : INT;
	CasKontrolyVystupnejBarieryP4 : TON;
	CasPoruchyServaSrobovaniaOsZ_M5 : TON;
	CasKontroly_KAM14 : TON;
END_VAR
```

### Program Logical/OdosielanieFotiek/FTP_CAM1 (IEC)
